  PROC DrawPart24()
    MoveL Offs(pOrigin,252.34,264.25,6.00),v60,z5,tPen\WObj:=wPaper;
    MoveL Offs(pOrigin,252.12,261.70,6.00),vTravel,z5,tPen\WObj:=wPaper;
    MoveL Offs(pOrigin,252.12,261.70,0.00),v60,z0,tPen\WObj:=wPaper;
    MoveL Offs(pOrigin,252.34,261.20,0.00),v40,z0,tPen\WObj:=wPaper;
    MoveL Offs(pOrigin,254.68,259.93,0.00),v40,z0,tPen\WObj:=wPaper;
    MoveL Offs(pOrigin,259.35,258.51,0.00),v40,z0,tPen\WObj:=wPaper;
    MoveL Offs(pOrigin,262.54,258.51,0.00),v40,fine,tPen\WObj:=wPaper;
    MoveL Offs(pOrigin,262.54,258.51,6.00),v60,z5,tPen\WObj:=wPaper;
    MoveL Offs(pOrigin,261.26,260.85,6.00),vTravel,z5,tPen\WObj:=wPaper;
    MoveL Offs(pOrigin,261.26,260.85,0.00),v60,z0,tPen\WObj:=wPaper;
    MoveL Offs(pOrigin,256.16,261.49,0.00),v40,z0,tPen\WObj:=wPaper;
    MoveL Offs(pOrigin,252.98,262.55,0.00),v40,z0,tPen\WObj:=wPaper;
    MoveL Offs(pOrigin,252.34,262.34,0.00),v40,z0,tPen\WObj:=wPaper;
    MoveL Offs(pOrigin,252.12,261.70,0.00),v40,fine,tPen\WObj:=wPaper;
    MoveL Offs(pOrigin,252.12,261.70,6.00),v60,z5,tPen\WObj:=wPaper;
    MoveL Offs(pOrigin,254.89,260.00,6.00),vTravel,z5,tPen\WObj:=wPaper;
    MoveL Offs(pOrigin,254.89,260.00,0.00),v60,z0,tPen\WObj:=wPaper;
    MoveL Offs(pOrigin,255.31,259.79,0.00),v40,z0,tPen\WObj:=wPaper;
    MoveL Offs(pOrigin,254.89,260.00,0.00),v40,fine,tPen\WObj:=wPaper;
    MoveL Offs(pOrigin,254.89,260.00,6.00),v60,z5,tPen\WObj:=wPaper;
    MoveL Offs(pOrigin,249.15,258.30,6.00),vTravel,z5,tPen\WObj:=wPaper;
    MoveL Offs(pOrigin,249.15,258.30,0.00),v60,z0,tPen\WObj:=wPaper;
    MoveL Offs(pOrigin,248.30,259.79,0.00),v40,z0,tPen\WObj:=wPaper;
    MoveL Offs(pOrigin,248.51,261.06,0.00),v40,fine,tPen\WObj:=wPaper;
    MoveL Offs(pOrigin,248.51,261.06,6.00),v60,z5,tPen\WObj:=wPaper;
    MoveL Offs(pOrigin,247.88,263.19,6.00),vTravel,z5,tPen\WObj:=wPaper;
    MoveL Offs(pOrigin,247.88,263.19,0.00),v60,z0,tPen\WObj:=wPaper;
    MoveL Offs(pOrigin,247.02,263.61,0.00),v40,z0,tPen\WObj:=wPaper;
    MoveL Offs(pOrigin,246.81,264.46,0.00),v40,z0,tPen\WObj:=wPaper;
    MoveL Offs(pOrigin,246.81,264.46,0.00),v40,z0,tPen\WObj:=wPaper;
    MoveL Offs(pOrigin,246.81,265.95,0.00),v40,z0,tPen\WObj:=wPaper;
    MoveL Offs(pOrigin,246.60,265.95,0.00),v40,z0,tPen\WObj:=wPaper;
    MoveL Offs(pOrigin,245.75,265.95,0.00),v40,z0,tPen\WObj:=wPaper;
    MoveL Offs(pOrigin,245.75,265.10,0.00),v40,z0,tPen\WObj:=wPaper;
    MoveL Offs(pOrigin,245.32,264.89,0.00),v40,z0,tPen\WObj:=wPaper;
    MoveL Offs(pOrigin,245.32,264.89,0.00),v40,z0,tPen\WObj:=wPaper;
    MoveL Offs(pOrigin,245.11,263.61,0.00),v40,z0,tPen\WObj:=wPaper;
    MoveL Offs(pOrigin,246.46,260.07,0.00),v40,z0,tPen\WObj:=wPaper;
    MoveL Offs(pOrigin,247.88,258.16,0.00),v40,z0,tPen\WObj:=wPaper;
    MoveL Offs(pOrigin,249.15,257.88,0.00),v40,fine,tPen\WObj:=wPaper;
    MoveL Offs(pOrigin,249.15,257.88,6.00),v60,z5,tPen\WObj:=wPaper;
    MoveL Offs(pOrigin,247.88,263.19,6.00),vTravel,z5,tPen\WObj:=wPaper;
    MoveL Offs(pOrigin,247.88,263.19,0.00),v60,z0,tPen\WObj:=wPaper;
    MoveL Offs(pOrigin,248.51,263.83,0.00),v40,fine,tPen\WObj:=wPaper;
    MoveL Offs(pOrigin,248.51,263.83,6.00),v60,z5,tPen\WObj:=wPaper;
    MoveL Offs(pOrigin,246.81,264.46,6.00),vTravel,z5,tPen\WObj:=wPaper;
    MoveL Offs(pOrigin,246.81,264.46,0.00),v60,z0,tPen\WObj:=wPaper;
    MoveL Offs(pOrigin,245.75,264.89,0.00),v40,z0,tPen\WObj:=wPaper;
    MoveL Offs(pOrigin,245.32,264.89,0.00),v40,z0,tPen\WObj:=wPaper;
    MoveL Offs(pOrigin,244.69,266.16,0.00),v40,z0,tPen\WObj:=wPaper;
    MoveL Offs(pOrigin,244.69,266.16,0.00),v40,z0,tPen\WObj:=wPaper;
    MoveL Offs(pOrigin,246.39,266.02,0.00),v40,z0,tPen\WObj:=wPaper;
    MoveL Offs(pOrigin,246.60,267.86,0.00),v40,z0,tPen\WObj:=wPaper;
    MoveL Offs(pOrigin,246.60,267.86,0.00),v40,z0,tPen\WObj:=wPaper;
    MoveL Offs(pOrigin,246.81,269.14,0.00),v40,z0,tPen\WObj:=wPaper;
    MoveL Offs(pOrigin,246.81,269.14,0.00),v40,z0,tPen\WObj:=wPaper;
    MoveL Offs(pOrigin,246.81,270.20,0.00),v40,z0,tPen\WObj:=wPaper;
    MoveL Offs(pOrigin,246.81,270.20,0.00),v40,z0,tPen\WObj:=wPaper;
    MoveL Offs(pOrigin,245.32,270.13,0.00),v40,z0,tPen\WObj:=wPaper;
    MoveL Offs(pOrigin,245.11,269.77,0.00),v40,z0,tPen\WObj:=wPaper;
    MoveL Offs(pOrigin,245.32,268.92,0.00),v40,z0,tPen\WObj:=wPaper;
    MoveL Offs(pOrigin,245.32,268.92,0.00),v40,z0,tPen\WObj:=wPaper;
    MoveL Offs(pOrigin,244.26,267.86,0.00),v40,z0,tPen\WObj:=wPaper;
    MoveL Offs(pOrigin,241.50,267.86,0.00),v40,z0,tPen\WObj:=wPaper;
    MoveL Offs(pOrigin,237.46,267.15,0.00),v40,z0,tPen\WObj:=wPaper;
    MoveL Offs(pOrigin,236.40,267.86,0.00),v40,z0,tPen\WObj:=wPaper;
    MoveL Offs(pOrigin,236.61,271.05,0.00),v40,z0,tPen\WObj:=wPaper;
    MoveL Offs(pOrigin,236.19,271.48,0.00),v40,fine,tPen\WObj:=wPaper;
    MoveL Offs(pOrigin,236.19,271.48,6.00),v60,z5,tPen\WObj:=wPaper;
    MoveL Offs(pOrigin,233.21,271.48,6.00),vTravel,z5,tPen\WObj:=wPaper;
    MoveL Offs(pOrigin,233.21,271.48,0.00),v60,z0,tPen\WObj:=wPaper;
    MoveL Offs(pOrigin,231.94,271.90,0.00),v40,z0,tPen\WObj:=wPaper;
    MoveL Offs(pOrigin,231.30,271.26,0.00),v40,z0,tPen\WObj:=wPaper;
    MoveL Offs(pOrigin,231.51,270.84,0.00),v40,z0,tPen\WObj:=wPaper;
    MoveL Offs(pOrigin,231.65,269.77,0.00),v40,z0,tPen\WObj:=wPaper;
    MoveL Offs(pOrigin,230.45,268.71,0.00),v40,z0,tPen\WObj:=wPaper;
    MoveL Offs(pOrigin,230.45,268.71,0.00),v40,z0,tPen\WObj:=wPaper;
    MoveL Offs(pOrigin,231.09,268.08,0.00),v40,z0,tPen\WObj:=wPaper;
    MoveL Offs(pOrigin,232.15,268.08,0.00),v40,z0,tPen\WObj:=wPaper;
    MoveL Offs(pOrigin,232.79,268.50,0.00),v40,z0,tPen\WObj:=wPaper;
    MoveL Offs(pOrigin,232.79,269.14,0.00),v40,z0,tPen\WObj:=wPaper;
    MoveL Offs(pOrigin,231.73,269.56,0.00),v40,fine,tPen\WObj:=wPaper;
    MoveL Offs(pOrigin,231.73,269.56,6.00),v60,z5,tPen\WObj:=wPaper;
    MoveL Offs(pOrigin,231.51,270.84,6.00),vTravel,z5,tPen\WObj:=wPaper;
    MoveL Offs(pOrigin,231.51,270.84,0.00),v60,z0,tPen\WObj:=wPaper;
    MoveL Offs(pOrigin,233.21,270.84,0.00),v40,z0,tPen\WObj:=wPaper;
    MoveL Offs(pOrigin,233.21,270.84,0.00),v40,z0,tPen\WObj:=wPaper;
    MoveL Offs(pOrigin,233.00,268.57,0.00),v40,z0,tPen\WObj:=wPaper;
    MoveL Offs(pOrigin,234.06,268.22,0.00),v40,z0,tPen\WObj:=wPaper;
    MoveL Offs(pOrigin,235.48,269.14,0.00),v40,z0,tPen\WObj:=wPaper;
    MoveL Offs(pOrigin,236.19,271.90,0.00),v40,z0,tPen\WObj:=wPaper;
    MoveL Offs(pOrigin,236.19,275.30,0.00),v40,fine,tPen\WObj:=wPaper;
    MoveL Offs(pOrigin,236.19,275.30,6.00),v60,z5,tPen\WObj:=wPaper;
    MoveL Offs(pOrigin,231.73,271.90,6.00),vTravel,z5,tPen\WObj:=wPaper;
    MoveL Offs(pOrigin,231.73,271.90,0.00),v60,z0,tPen\WObj:=wPaper;
    MoveL Offs(pOrigin,230.88,271.26,0.00),v40,z0,tPen\WObj:=wPaper;
    MoveL Offs(pOrigin,226.41,271.69,0.00),v40,z0,tPen\WObj:=wPaper;
    MoveL Offs(pOrigin,217.49,270.41,0.00),v40,z0,tPen\WObj:=wPaper;
    MoveL Offs(pOrigin,217.13,270.62,0.00),v40,z0,tPen\WObj:=wPaper;
    MoveL Offs(pOrigin,217.27,271.05,0.00),v40,z0,tPen\WObj:=wPaper;
    MoveL Offs(pOrigin,217.06,270.41,0.00),v40,z0,tPen\WObj:=wPaper;
    MoveL Offs(pOrigin,214.30,268.57,0.00),v40,z0,tPen\WObj:=wPaper;
    MoveL Offs(pOrigin,213.88,267.86,0.00),v40,z0,tPen\WObj:=wPaper;
    MoveL Offs(pOrigin,213.88,267.86,0.00),v40,z0,tPen\WObj:=wPaper;
    MoveL Offs(pOrigin,214.73,267.65,0.00),v40,z0,tPen\WObj:=wPaper;
    MoveL Offs(pOrigin,215.15,268.71,0.00),v40,z0,tPen\WObj:=wPaper;
    MoveL Offs(pOrigin,215.15,268.08,0.00),v40,z0,tPen\WObj:=wPaper;
    MoveL Offs(pOrigin,219.19,268.50,0.00),v40,z0,tPen\WObj:=wPaper;
    MoveL Offs(pOrigin,219.19,268.50,0.00),v40,z0,tPen\WObj:=wPaper;
    MoveL Offs(pOrigin,222.38,268.92,0.00),v40,z0,tPen\WObj:=wPaper;
    MoveL Offs(pOrigin,222.38,268.92,0.00),v40,z0,tPen\WObj:=wPaper;
    MoveL Offs(pOrigin,225.56,269.14,0.00),v40,z0,tPen\WObj:=wPaper;
    MoveL Offs(pOrigin,225.56,269.14,0.00),v40,z0,tPen\WObj:=wPaper;
    MoveL Offs(pOrigin,228.96,269.35,0.00),v40,z0,tPen\WObj:=wPaper;
    MoveL Offs(pOrigin,229.81,268.71,0.00),v40,z0,tPen\WObj:=wPaper;
    MoveL Offs(pOrigin,230.45,268.71,0.00),v40,z0,tPen\WObj:=wPaper;
    MoveL Offs(pOrigin,229.60,268.50,0.00),v40,z0,tPen\WObj:=wPaper;
    MoveL Offs(pOrigin,229.18,267.65,0.00),v40,z0,tPen\WObj:=wPaper;
    MoveL Offs(pOrigin,229.18,267.65,0.00),v40,z0,tPen\WObj:=wPaper;
    MoveL Offs(pOrigin,225.14,267.44,0.00),v40,z0,tPen\WObj:=wPaper;
  ENDPROC

  PROC DrawPart25()
    MoveL Offs(pOrigin,223.23,267.01,0.00),v40,z0,tPen\WObj:=wPaper;
    MoveL Offs(pOrigin,222.52,268.08,0.00),v40,z0,tPen\WObj:=wPaper;
    MoveL Offs(pOrigin,225.56,268.50,0.00),v40,z0,tPen\WObj:=wPaper;
    MoveL Offs(pOrigin,225.56,268.50,0.00),v40,z0,tPen\WObj:=wPaper;
    MoveL Offs(pOrigin,229.18,268.29,0.00),v40,z0,tPen\WObj:=wPaper;
    MoveL Offs(pOrigin,229.18,267.65,0.00),v40,z0,tPen\WObj:=wPaper;
    MoveL Offs(pOrigin,229.81,267.01,0.00),v40,z0,tPen\WObj:=wPaper;
    MoveL Offs(pOrigin,229.81,267.01,0.00),v40,z0,tPen\WObj:=wPaper;
    MoveL Offs(pOrigin,229.18,266.59,0.00),v40,z0,tPen\WObj:=wPaper;
    MoveL Offs(pOrigin,228.11,266.59,0.00),v40,z0,tPen\WObj:=wPaper;
    MoveL Offs(pOrigin,222.38,264.75,0.00),v40,z0,tPen\WObj:=wPaper;
    MoveL Offs(pOrigin,220.46,263.90,0.00),v40,z0,tPen\WObj:=wPaper;
    MoveL Offs(pOrigin,218.76,262.76,0.00),v40,z0,tPen\WObj:=wPaper;
    MoveL Offs(pOrigin,218.34,262.12,0.00),v40,z0,tPen\WObj:=wPaper;
    MoveL Offs(pOrigin,218.34,262.12,0.00),v40,z0,tPen\WObj:=wPaper;
    MoveL Offs(pOrigin,217.06,261.49,0.00),v40,z0,tPen\WObj:=wPaper;
    MoveL Offs(pOrigin,216.21,259.58,0.00),v40,z0,tPen\WObj:=wPaper;
    MoveL Offs(pOrigin,216.21,259.58,0.00),v40,z0,tPen\WObj:=wPaper;
    MoveL Offs(pOrigin,217.27,259.15,0.00),v40,z0,tPen\WObj:=wPaper;
    MoveL Offs(pOrigin,218.55,259.93,0.00),v40,z0,tPen\WObj:=wPaper;
    MoveL Offs(pOrigin,219.82,260.00,0.00),v40,z0,tPen\WObj:=wPaper;
    MoveL Offs(pOrigin,219.82,260.00,0.00),v40,z0,tPen\WObj:=wPaper;
    MoveL Offs(pOrigin,219.82,260.64,0.00),v40,z0,tPen\WObj:=wPaper;
    MoveL Offs(pOrigin,220.68,260.64,0.00),v40,z0,tPen\WObj:=wPaper;
    MoveL Offs(pOrigin,220.68,260.64,0.00),v40,z0,tPen\WObj:=wPaper;
    MoveL Offs(pOrigin,220.46,259.79,0.00),v40,z0,tPen\WObj:=wPaper;
    MoveL Offs(pOrigin,219.82,260.00,0.00),v40,z0,tPen\WObj:=wPaper;
    MoveL Offs(pOrigin,220.68,259.79,0.00),v40,z0,tPen\WObj:=wPaper;
    MoveL Offs(pOrigin,222.80,259.36,0.00),v40,z0,tPen\WObj:=wPaper;
    MoveL Offs(pOrigin,223.01,260.42,0.00),v40,z0,tPen\WObj:=wPaper;
    MoveL Offs(pOrigin,221.10,260.71,0.00),v40,z0,tPen\WObj:=wPaper;
    MoveL Offs(pOrigin,220.89,261.49,0.00),v40,z0,tPen\WObj:=wPaper;
    MoveL Offs(pOrigin,221.10,261.91,0.00),v40,z0,tPen\WObj:=wPaper;
    MoveL Offs(pOrigin,222.80,262.83,0.00),v40,z0,tPen\WObj:=wPaper;
    MoveL Offs(pOrigin,223.08,262.20,0.00),v40,z0,tPen\WObj:=wPaper;
    MoveL Offs(pOrigin,224.07,261.49,0.00),v40,z0,tPen\WObj:=wPaper;
    MoveL Offs(pOrigin,224.07,260.85,0.00),v40,z0,tPen\WObj:=wPaper;
    MoveL Offs(pOrigin,225.99,260.64,0.00),v40,z0,tPen\WObj:=wPaper;
    MoveL Offs(pOrigin,226.20,261.06,0.00),v40,z0,tPen\WObj:=wPaper;
    MoveL Offs(pOrigin,226.20,261.06,0.00),v40,z0,tPen\WObj:=wPaper;
    MoveL Offs(pOrigin,227.05,261.27,0.00),v40,z0,tPen\WObj:=wPaper;
    MoveL Offs(pOrigin,227.69,262.12,0.00),v40,z0,tPen\WObj:=wPaper;
    MoveL Offs(pOrigin,227.69,263.40,0.00),v40,fine,tPen\WObj:=wPaper;
    MoveL Offs(pOrigin,227.69,263.40,6.00),v60,z5,tPen\WObj:=wPaper;
    MoveL Offs(pOrigin,227.90,262.12,6.00),vTravel,z5,tPen\WObj:=wPaper;
    MoveL Offs(pOrigin,227.90,262.12,0.00),v60,z0,tPen\WObj:=wPaper;
    MoveL Offs(pOrigin,228.96,261.91,0.00),v40,z0,tPen\WObj:=wPaper;
    MoveL Offs(pOrigin,228.96,261.91,0.00),v40,z0,tPen\WObj:=wPaper;
    MoveL Offs(pOrigin,229.60,263.61,0.00),v40,z0,tPen\WObj:=wPaper;
    MoveL Offs(pOrigin,230.88,263.26,0.00),v40,z0,tPen\WObj:=wPaper;
    MoveL Offs(pOrigin,231.51,262.34,0.00),v40,z0,tPen\WObj:=wPaper;
    MoveL Offs(pOrigin,231.51,262.34,0.00),v40,z0,tPen\WObj:=wPaper;
    MoveL Offs(pOrigin,233.21,262.12,0.00),v40,z0,tPen\WObj:=wPaper;
    MoveL Offs(pOrigin,233.21,262.12,0.00),v40,z0,tPen\WObj:=wPaper;
    MoveL Offs(pOrigin,233.64,262.98,0.00),v40,fine,tPen\WObj:=wPaper;
    MoveL Offs(pOrigin,233.64,262.98,6.00),v60,z5,tPen\WObj:=wPaper;
    MoveL Offs(pOrigin,233.85,264.46,6.00),vTravel,z5,tPen\WObj:=wPaper;
    MoveL Offs(pOrigin,233.85,264.46,0.00),v60,z0,tPen\WObj:=wPaper;
    MoveL Offs(pOrigin,234.84,263.54,0.00),v40,z0,tPen\WObj:=wPaper;
    MoveL Offs(pOrigin,234.91,262.83,0.00),v40,z0,tPen\WObj:=wPaper;
    MoveL Offs(pOrigin,233.85,262.98,0.00),v40,z0,tPen\WObj:=wPaper;
    MoveL Offs(pOrigin,233.28,263.61,0.00),v40,z0,tPen\WObj:=wPaper;
    MoveL Offs(pOrigin,233.21,264.46,0.00),v40,z0,tPen\WObj:=wPaper;
    MoveL Offs(pOrigin,233.21,264.46,0.00),v40,z0,tPen\WObj:=wPaper;
    MoveL Offs(pOrigin,234.27,264.89,0.00),v40,z0,tPen\WObj:=wPaper;
    MoveL Offs(pOrigin,235.34,265.95,0.00),v40,z0,tPen\WObj:=wPaper;
    MoveL Offs(pOrigin,235.27,267.23,0.00),v40,z0,tPen\WObj:=wPaper;
    MoveL Offs(pOrigin,234.27,268.08,0.00),v40,z0,tPen\WObj:=wPaper;
    MoveL Offs(pOrigin,233.85,268.08,0.00),v40,z0,tPen\WObj:=wPaper;
    MoveL Offs(pOrigin,233.14,266.87,0.00),v40,z0,tPen\WObj:=wPaper;
    MoveL Offs(pOrigin,231.51,266.59,0.00),v40,z0,tPen\WObj:=wPaper;
    MoveL Offs(pOrigin,231.51,266.59,0.00),v40,z0,tPen\WObj:=wPaper;
    MoveL Offs(pOrigin,230.45,267.01,0.00),v40,z0,tPen\WObj:=wPaper;
    MoveL Offs(pOrigin,230.45,267.01,0.00),v40,z0,tPen\WObj:=wPaper;
    MoveL Offs(pOrigin,230.66,268.08,0.00),v40,fine,tPen\WObj:=wPaper;
    MoveL Offs(pOrigin,230.66,268.08,6.00),v60,z5,tPen\WObj:=wPaper;
    MoveL Offs(pOrigin,231.51,266.59,6.00),vTravel,z5,tPen\WObj:=wPaper;
    MoveL Offs(pOrigin,231.51,266.59,0.00),v60,z0,tPen\WObj:=wPaper;
    MoveL Offs(pOrigin,232.36,265.74,0.00),v40,z0,tPen\WObj:=wPaper;
    MoveL Offs(pOrigin,232.79,264.46,0.00),v40,z0,tPen\WObj:=wPaper;
    MoveL Offs(pOrigin,232.79,264.46,0.00),v40,z0,tPen\WObj:=wPaper;
    MoveL Offs(pOrigin,232.15,264.25,0.00),v40,z0,tPen\WObj:=wPaper;
    MoveL Offs(pOrigin,230.45,264.89,0.00),v40,z0,tPen\WObj:=wPaper;
    MoveL Offs(pOrigin,230.38,264.89,0.00),v40,z0,tPen\WObj:=wPaper;
    MoveL Offs(pOrigin,230.17,265.45,0.00),v40,z0,tPen\WObj:=wPaper;
    MoveL Offs(pOrigin,229.39,265.74,0.00),v40,z0,tPen\WObj:=wPaper;
    MoveL Offs(pOrigin,228.40,265.52,0.00),v40,z0,tPen\WObj:=wPaper;
    MoveL Offs(pOrigin,228.96,264.89,0.00),v40,z0,tPen\WObj:=wPaper;
    MoveL Offs(pOrigin,229.81,264.67,0.00),v40,z0,tPen\WObj:=wPaper;
    MoveL Offs(pOrigin,230.38,264.89,0.00),v40,fine,tPen\WObj:=wPaper;
    MoveL Offs(pOrigin,230.38,264.89,6.00),v60,z5,tPen\WObj:=wPaper;
    MoveL Offs(pOrigin,228.32,265.10,6.00),vTravel,z5,tPen\WObj:=wPaper;
    MoveL Offs(pOrigin,228.32,265.10,0.00),v60,z0,tPen\WObj:=wPaper;
    MoveL Offs(pOrigin,226.84,265.10,0.00),v40,z0,tPen\WObj:=wPaper;
    MoveL Offs(pOrigin,226.41,265.74,0.00),v40,fine,tPen\WObj:=wPaper;
    MoveL Offs(pOrigin,226.41,265.74,6.00),v60,z5,tPen\WObj:=wPaper;
    MoveL Offs(pOrigin,222.80,267.01,6.00),vTravel,z5,tPen\WObj:=wPaper;
    MoveL Offs(pOrigin,222.80,267.01,0.00),v60,z0,tPen\WObj:=wPaper;
    MoveL Offs(pOrigin,221.74,266.80,0.00),v40,z0,tPen\WObj:=wPaper;
    MoveL Offs(pOrigin,221.52,267.23,0.00),v40,z0,tPen\WObj:=wPaper;
    MoveL Offs(pOrigin,221.52,267.23,0.00),v40,z0,tPen\WObj:=wPaper;
    MoveL Offs(pOrigin,217.49,266.09,0.00),v40,z0,tPen\WObj:=wPaper;
    MoveL Offs(pOrigin,215.15,264.67,0.00),v40,z0,tPen\WObj:=wPaper;
    MoveL Offs(pOrigin,214.73,263.90,0.00),v40,z0,tPen\WObj:=wPaper;
    MoveL Offs(pOrigin,213.88,263.68,0.00),v40,z0,tPen\WObj:=wPaper;
    MoveL Offs(pOrigin,213.24,262.98,0.00),v40,z0,tPen\WObj:=wPaper;
    MoveL Offs(pOrigin,213.24,262.98,0.00),v40,z0,tPen\WObj:=wPaper;
    MoveL Offs(pOrigin,212.67,260.42,0.00),v40,z0,tPen\WObj:=wPaper;
    MoveL Offs(pOrigin,214.51,259.15,0.00),v40,z0,tPen\WObj:=wPaper;
    MoveL Offs(pOrigin,214.51,259.15,0.00),v40,z0,tPen\WObj:=wPaper;
    MoveL Offs(pOrigin,213.66,258.51,0.00),v40,z0,tPen\WObj:=wPaper;
    MoveL Offs(pOrigin,211.75,258.51,0.00),v40,fine,tPen\WObj:=wPaper;
    MoveL Offs(pOrigin,211.75,258.51,6.00),v60,z5,tPen\WObj:=wPaper;
    MoveL Offs(pOrigin,213.45,256.60,6.00),vTravel,z5,tPen\WObj:=wPaper;
    MoveL Offs(pOrigin,213.45,256.60,0.00),v60,z0,tPen\WObj:=wPaper;
    MoveL Offs(pOrigin,214.73,257.45,0.00),v40,z0,tPen\WObj:=wPaper;
    MoveL Offs(pOrigin,215.36,259.15,0.00),v40,z0,tPen\WObj:=wPaper;
    MoveL Offs(pOrigin,215.36,259.15,0.00),v40,z0,tPen\WObj:=wPaper;
    MoveL Offs(pOrigin,216.21,259.58,0.00),v40,fine,tPen\WObj:=wPaper;
    MoveL Offs(pOrigin,216.21,259.58,6.00),v60,z5,tPen\WObj:=wPaper;
  ENDPROC

  PROC DrawPart26()
    MoveL Offs(pOrigin,217.91,259.58,6.00),vTravel,z5,tPen\WObj:=wPaper;
    MoveL Offs(pOrigin,217.91,259.58,0.00),v60,z0,tPen\WObj:=wPaper;
    MoveL Offs(pOrigin,218.34,260.00,0.00),v40,z0,tPen\WObj:=wPaper;
    MoveL Offs(pOrigin,217.91,259.58,0.00),v40,fine,tPen\WObj:=wPaper;
    MoveL Offs(pOrigin,217.91,259.58,6.00),v60,z5,tPen\WObj:=wPaper;
    MoveL Offs(pOrigin,216.85,261.49,6.00),vTravel,z5,tPen\WObj:=wPaper;
    MoveL Offs(pOrigin,216.85,261.49,0.00),v60,z0,tPen\WObj:=wPaper;
    MoveL Offs(pOrigin,217.27,261.91,0.00),v40,z0,tPen\WObj:=wPaper;
    MoveL Offs(pOrigin,216.85,261.49,0.00),v40,fine,tPen\WObj:=wPaper;
    MoveL Offs(pOrigin,216.85,261.49,6.00),v60,z5,tPen\WObj:=wPaper;
    MoveL Offs(pOrigin,215.79,265.31,6.00),vTravel,z5,tPen\WObj:=wPaper;
    MoveL Offs(pOrigin,215.79,265.31,0.00),v60,z0,tPen\WObj:=wPaper;
    MoveL Offs(pOrigin,216.21,265.52,0.00),v40,z0,tPen\WObj:=wPaper;
    MoveL Offs(pOrigin,215.79,265.31,0.00),v40,fine,tPen\WObj:=wPaper;
    MoveL Offs(pOrigin,215.79,265.31,6.00),v60,z5,tPen\WObj:=wPaper;
    MoveL Offs(pOrigin,213.88,267.86,6.00),vTravel,z5,tPen\WObj:=wPaper;
    MoveL Offs(pOrigin,213.88,267.86,0.00),v60,z0,tPen\WObj:=wPaper;
    MoveL Offs(pOrigin,209.41,266.30,0.00),v40,z0,tPen\WObj:=wPaper;
    MoveL Offs(pOrigin,208.77,265.17,0.00),v40,z0,tPen\WObj:=wPaper;
    MoveL Offs(pOrigin,207.57,264.67,0.00),v40,z0,tPen\WObj:=wPaper;
    MoveL Offs(pOrigin,207.29,263.61,0.00),v40,z0,tPen\WObj:=wPaper;
    MoveL Offs(pOrigin,207.29,263.61,0.00),v40,z0,tPen\WObj:=wPaper;
    MoveL Offs(pOrigin,204.52,263.12,0.00),v40,z0,tPen\WObj:=wPaper;
    MoveL Offs(pOrigin,204.10,261.91,0.00),v40,z0,tPen\WObj:=wPaper;
    MoveL Offs(pOrigin,204.10,261.91,0.00),v40,z0,tPen\WObj:=wPaper;
    MoveL Offs(pOrigin,207.07,260.92,0.00),v40,z0,tPen\WObj:=wPaper;
    MoveL Offs(pOrigin,207.29,263.61,0.00),v40,fine,tPen\WObj:=wPaper;
    MoveL Offs(pOrigin,207.29,263.61,6.00),v60,z5,tPen\WObj:=wPaper;
    MoveL Offs(pOrigin,207.50,265.31,6.00),vTravel,z5,tPen\WObj:=wPaper;
    MoveL Offs(pOrigin,207.50,265.31,0.00),v60,z0,tPen\WObj:=wPaper;
    MoveL Offs(pOrigin,206.65,265.95,0.00),v40,z0,tPen\WObj:=wPaper;
    MoveL Offs(pOrigin,206.23,270.84,0.00),v40,z0,tPen\WObj:=wPaper;
    MoveL Offs(pOrigin,205.38,272.33,0.00),v40,z0,tPen\WObj:=wPaper;
    MoveL Offs(pOrigin,205.30,274.45,0.00),v40,z0,tPen\WObj:=wPaper;
    MoveL Offs(pOrigin,204.74,275.09,0.00),v40,z0,tPen\WObj:=wPaper;
    MoveL Offs(pOrigin,204.88,276.72,0.00),v40,z0,tPen\WObj:=wPaper;
    MoveL Offs(pOrigin,204.31,277.21,0.00),v40,z0,tPen\WObj:=wPaper;
    MoveL Offs(pOrigin,204.52,279.12,0.00),v40,z0,tPen\WObj:=wPaper;
    MoveL Offs(pOrigin,204.52,279.12,0.00),v40,z0,tPen\WObj:=wPaper;
    MoveL Offs(pOrigin,203.75,279.76,0.00),v40,z0,tPen\WObj:=wPaper;
    MoveL Offs(pOrigin,203.53,280.83,0.00),v40,z0,tPen\WObj:=wPaper;
    MoveL Offs(pOrigin,204.17,281.46,0.00),v40,z0,tPen\WObj:=wPaper;
    MoveL Offs(pOrigin,204.74,282.95,0.00),v40,z0,tPen\WObj:=wPaper;
    MoveL Offs(pOrigin,204.95,284.86,0.00),v40,z0,tPen\WObj:=wPaper;
    MoveL Offs(pOrigin,204.74,286.56,0.00),v40,z0,tPen\WObj:=wPaper;
    MoveL Offs(pOrigin,204.74,286.56,0.00),v40,z0,tPen\WObj:=wPaper;
    MoveL Offs(pOrigin,205.45,289.11,0.00),v40,z0,tPen\WObj:=wPaper;
    MoveL Offs(pOrigin,206.65,290.17,0.00),v40,z0,tPen\WObj:=wPaper;
    MoveL Offs(pOrigin,206.23,291.24,0.00),v40,z0,tPen\WObj:=wPaper;
    MoveL Offs(pOrigin,206.23,291.24,0.00),v40,z0,tPen\WObj:=wPaper;
    MoveL Offs(pOrigin,206.23,293.15,0.00),v40,fine,tPen\WObj:=wPaper;
    MoveL Offs(pOrigin,206.23,293.15,6.00),v60,z5,tPen\WObj:=wPaper;
    MoveL Offs(pOrigin,206.23,291.24,6.00),vTravel,z5,tPen\WObj:=wPaper;
    MoveL Offs(pOrigin,206.23,291.24,0.00),v60,z0,tPen\WObj:=wPaper;
    MoveL Offs(pOrigin,205.38,290.81,0.00),v40,z0,tPen\WObj:=wPaper;
    MoveL Offs(pOrigin,205.16,290.17,0.00),v40,z0,tPen\WObj:=wPaper;
    MoveL Offs(pOrigin,205.38,289.33,0.00),v40,z0,tPen\WObj:=wPaper;
    MoveL Offs(pOrigin,205.80,289.54,0.00),v40,z0,tPen\WObj:=wPaper;
    MoveL Offs(pOrigin,206.23,289.75,0.00),v40,z0,tPen\WObj:=wPaper;
    MoveL Offs(pOrigin,205.80,289.54,0.00),v40,fine,tPen\WObj:=wPaper;
    MoveL Offs(pOrigin,205.80,289.54,6.00),v60,z5,tPen\WObj:=wPaper;
    MoveL Offs(pOrigin,202.40,289.96,6.00),vTravel,z5,tPen\WObj:=wPaper;
    MoveL Offs(pOrigin,202.40,289.96,0.00),v60,z0,tPen\WObj:=wPaper;
    MoveL Offs(pOrigin,202.40,289.11,0.00),v40,z0,tPen\WObj:=wPaper;
    MoveL Offs(pOrigin,201.55,288.69,0.00),v40,z0,tPen\WObj:=wPaper;
    MoveL Offs(pOrigin,201.55,288.69,0.00),v40,z0,tPen\WObj:=wPaper;
    MoveL Offs(pOrigin,200.35,286.14,0.00),v40,z0,tPen\WObj:=wPaper;
    MoveL Offs(pOrigin,199.21,284.79,0.00),v40,z0,tPen\WObj:=wPaper;
    MoveL Offs(pOrigin,198.36,284.44,0.00),v40,z0,tPen\WObj:=wPaper;
    MoveL Offs(pOrigin,197.37,285.29,0.00),v40,z0,tPen\WObj:=wPaper;
    MoveL Offs(pOrigin,197.30,286.14,0.00),v40,z0,tPen\WObj:=wPaper;
    MoveL Offs(pOrigin,197.30,286.14,0.00),v40,z0,tPen\WObj:=wPaper;
    MoveL Offs(pOrigin,197.44,287.20,0.00),v40,z0,tPen\WObj:=wPaper;
    MoveL Offs(pOrigin,199.07,289.96,0.00),v40,z0,tPen\WObj:=wPaper;
    MoveL Offs(pOrigin,199.43,291.45,0.00),v40,z0,tPen\WObj:=wPaper;
    MoveL Offs(pOrigin,199.43,291.45,0.00),v40,z0,tPen\WObj:=wPaper;
    MoveL Offs(pOrigin,198.01,290.81,0.00),v40,z0,tPen\WObj:=wPaper;
    MoveL Offs(pOrigin,195.74,286.35,0.00),v40,z0,tPen\WObj:=wPaper;
    MoveL Offs(pOrigin,195.18,285.92,0.00),v40,z0,tPen\WObj:=wPaper;
    MoveL Offs(pOrigin,195.18,285.92,0.00),v40,z0,tPen\WObj:=wPaper;
    MoveL Offs(pOrigin,194.54,287.20,0.00),v40,z0,tPen\WObj:=wPaper;
    MoveL Offs(pOrigin,193.90,287.20,0.00),v40,z0,tPen\WObj:=wPaper;
    MoveL Offs(pOrigin,193.26,287.84,0.00),v40,z0,tPen\WObj:=wPaper;
    MoveL Offs(pOrigin,193.69,289.11,0.00),v40,z0,tPen\WObj:=wPaper;
    MoveL Offs(pOrigin,194.32,289.89,0.00),v40,z0,tPen\WObj:=wPaper;
    MoveL Offs(pOrigin,195.10,290.25,0.00),v40,z0,tPen\WObj:=wPaper;
    MoveL Offs(pOrigin,199.21,295.91,0.00),v40,z0,tPen\WObj:=wPaper;
    MoveL Offs(pOrigin,200.91,297.47,0.00),v40,z0,tPen\WObj:=wPaper;
    MoveL Offs(pOrigin,201.98,297.61,0.00),v40,z0,tPen\WObj:=wPaper;
    MoveL Offs(pOrigin,201.98,297.61,0.00),v40,z0,tPen\WObj:=wPaper;
    MoveL Offs(pOrigin,201.98,296.55,0.00),v40,z0,tPen\WObj:=wPaper;
    MoveL Offs(pOrigin,201.98,296.55,0.00),v40,z0,tPen\WObj:=wPaper;
    MoveL Offs(pOrigin,204.10,296.12,0.00),v40,z0,tPen\WObj:=wPaper;
    MoveL Offs(pOrigin,204.10,296.12,0.00),v40,z0,tPen\WObj:=wPaper;
    MoveL Offs(pOrigin,203.82,295.06,0.00),v40,z0,tPen\WObj:=wPaper;
    MoveL Offs(pOrigin,203.25,294.42,0.00),v40,z0,tPen\WObj:=wPaper;
    MoveL Offs(pOrigin,201.55,293.79,0.00),v40,z0,tPen\WObj:=wPaper;
    MoveL Offs(pOrigin,201.12,294.21,0.00),v40,z0,tPen\WObj:=wPaper;
    MoveL Offs(pOrigin,201.98,296.55,0.00),v40,z0,tPen\WObj:=wPaper;
    MoveL Offs(pOrigin,201.98,297.61,0.00),v40,z0,tPen\WObj:=wPaper;
    MoveL Offs(pOrigin,202.40,298.46,0.00),v40,fine,tPen\WObj:=wPaper;
    MoveL Offs(pOrigin,202.40,298.46,6.00),v60,z5,tPen\WObj:=wPaper;
    MoveL Offs(pOrigin,202.40,299.95,6.00),vTravel,z5,tPen\WObj:=wPaper;
    MoveL Offs(pOrigin,202.40,299.95,0.00),v60,z0,tPen\WObj:=wPaper;
    MoveL Offs(pOrigin,200.49,299.31,0.00),v40,z0,tPen\WObj:=wPaper;
    MoveL Offs(pOrigin,199.71,299.52,0.00),v40,z0,tPen\WObj:=wPaper;
    MoveL Offs(pOrigin,199.71,300.38,0.00),v40,z0,tPen\WObj:=wPaper;
    MoveL Offs(pOrigin,201.34,301.86,0.00),v40,z0,tPen\WObj:=wPaper;
    MoveL Offs(pOrigin,201.34,301.86,0.00),v40,z0,tPen\WObj:=wPaper;
    MoveL Offs(pOrigin,201.34,302.92,0.00),v40,z0,tPen\WObj:=wPaper;
    MoveL Offs(pOrigin,201.34,302.92,0.00),v40,z0,tPen\WObj:=wPaper;
    MoveL Offs(pOrigin,203.04,303.92,0.00),v40,z0,tPen\WObj:=wPaper;
    MoveL Offs(pOrigin,204.74,304.41,0.00),v40,fine,tPen\WObj:=wPaper;
    MoveL Offs(pOrigin,204.74,304.41,6.00),v60,z5,tPen\WObj:=wPaper;
    MoveL Offs(pOrigin,204.74,306.11,6.00),vTravel,z5,tPen\WObj:=wPaper;
    MoveL Offs(pOrigin,204.74,306.11,0.00),v60,z0,tPen\WObj:=wPaper;
    MoveL Offs(pOrigin,204.31,305.55,0.00),v40,z0,tPen\WObj:=wPaper;
    MoveL Offs(pOrigin,200.27,304.27,0.00),v40,z0,tPen\WObj:=wPaper;
    MoveL Offs(pOrigin,198.36,302.71,0.00),v40,z0,tPen\WObj:=wPaper;
    MoveL Offs(pOrigin,196.66,301.86,0.00),v40,z0,tPen\WObj:=wPaper;
  ENDPROC

  PROC DrawPart27()
    MoveL Offs(pOrigin,194.47,298.46,0.00),v40,z0,tPen\WObj:=wPaper;
    MoveL Offs(pOrigin,193.90,298.04,0.00),v40,z0,tPen\WObj:=wPaper;
    MoveL Offs(pOrigin,193.90,298.04,0.00),v40,z0,tPen\WObj:=wPaper;
    MoveL Offs(pOrigin,193.69,298.67,0.00),v40,z0,tPen\WObj:=wPaper;
    MoveL Offs(pOrigin,194.68,301.44,0.00),v40,z0,tPen\WObj:=wPaper;
    MoveL Offs(pOrigin,196.88,304.84,0.00),v40,z0,tPen\WObj:=wPaper;
    MoveL Offs(pOrigin,200.06,306.47,0.00),v40,z0,tPen\WObj:=wPaper;
    MoveL Offs(pOrigin,200.91,306.25,0.00),v40,z0,tPen\WObj:=wPaper;
    MoveL Offs(pOrigin,203.25,306.75,0.00),v40,z0,tPen\WObj:=wPaper;
    MoveL Offs(pOrigin,203.25,306.75,0.00),v40,z0,tPen\WObj:=wPaper;
    MoveL Offs(pOrigin,204.10,307.81,0.00),v40,z0,tPen\WObj:=wPaper;
    MoveL Offs(pOrigin,203.89,308.45,0.00),v40,z0,tPen\WObj:=wPaper;
    MoveL Offs(pOrigin,204.52,307.81,0.00),v40,z0,tPen\WObj:=wPaper;
    MoveL Offs(pOrigin,206.86,307.60,0.00),v40,fine,tPen\WObj:=wPaper;
    MoveL Offs(pOrigin,206.86,307.60,6.00),v60,z5,tPen\WObj:=wPaper;
    MoveL Offs(pOrigin,208.35,306.11,6.00),vTravel,z5,tPen\WObj:=wPaper;
    MoveL Offs(pOrigin,208.35,306.11,0.00),v60,z0,tPen\WObj:=wPaper;
    MoveL Offs(pOrigin,204.74,306.11,0.00),v40,z0,tPen\WObj:=wPaper;
    MoveL Offs(pOrigin,204.74,306.11,0.00),v40,z0,tPen\WObj:=wPaper;
    MoveL Offs(pOrigin,203.68,306.33,0.00),v40,z0,tPen\WObj:=wPaper;
    MoveL Offs(pOrigin,203.25,306.75,0.00),v40,fine,tPen\WObj:=wPaper;
    MoveL Offs(pOrigin,203.25,306.75,6.00),v60,z5,tPen\WObj:=wPaper;
    MoveL Offs(pOrigin,204.74,309.09,6.00),vTravel,z5,tPen\WObj:=wPaper;
    MoveL Offs(pOrigin,204.74,309.09,0.00),v60,z0,tPen\WObj:=wPaper;
    MoveL Offs(pOrigin,205.38,309.94,0.00),v40,z0,tPen\WObj:=wPaper;
    MoveL Offs(pOrigin,205.38,309.94,0.00),v40,z0,tPen\WObj:=wPaper;
    MoveL Offs(pOrigin,203.68,308.52,0.00),v40,z0,tPen\WObj:=wPaper;
    MoveL Offs(pOrigin,200.27,308.24,0.00),v40,z0,tPen\WObj:=wPaper;
    MoveL Offs(pOrigin,197.73,307.32,0.00),v40,z0,tPen\WObj:=wPaper;
    MoveL Offs(pOrigin,195.18,305.69,0.00),v40,z0,tPen\WObj:=wPaper;
    MoveL Offs(pOrigin,194.32,304.20,0.00),v40,z0,tPen\WObj:=wPaper;
    MoveL Offs(pOrigin,193.90,303.99,0.00),v40,z0,tPen\WObj:=wPaper;
    MoveL Offs(pOrigin,193.90,303.99,0.00),v40,z0,tPen\WObj:=wPaper;
    MoveL Offs(pOrigin,193.26,300.16,0.00),v40,fine,tPen\WObj:=wPaper;
    MoveL Offs(pOrigin,193.26,300.16,6.00),v60,z5,tPen\WObj:=wPaper;
    MoveL Offs(pOrigin,191.35,300.80,6.00),vTravel,z5,tPen\WObj:=wPaper;
    MoveL Offs(pOrigin,191.35,300.80,0.00),v60,z0,tPen\WObj:=wPaper;
    MoveL Offs(pOrigin,191.35,296.98,0.00),v40,z0,tPen\WObj:=wPaper;
    MoveL Offs(pOrigin,192.41,293.58,0.00),v40,z0,tPen\WObj:=wPaper;
    MoveL Offs(pOrigin,191.63,292.73,0.00),v40,z0,tPen\WObj:=wPaper;
    MoveL Offs(pOrigin,191.49,291.95,0.00),v40,z0,tPen\WObj:=wPaper;
    MoveL Offs(pOrigin,190.93,291.66,0.00),v40,z0,tPen\WObj:=wPaper;
    MoveL Offs(pOrigin,190.93,291.66,0.00),v40,z0,tPen\WObj:=wPaper;
    MoveL Offs(pOrigin,190.22,292.73,0.00),v40,z0,tPen\WObj:=wPaper;
    MoveL Offs(pOrigin,189.44,295.70,0.00),v40,z0,tPen\WObj:=wPaper;
    MoveL Offs(pOrigin,189.23,297.83,0.00),v40,z0,tPen\WObj:=wPaper;
    MoveL Offs(pOrigin,189.65,299.52,0.00),v40,z0,tPen\WObj:=wPaper;
    MoveL Offs(pOrigin,189.65,299.52,0.00),v40,z0,tPen\WObj:=wPaper;
    MoveL Offs(pOrigin,190.43,302.50,0.00),v40,z0,tPen\WObj:=wPaper;
    MoveL Offs(pOrigin,192.13,305.90,0.00),v40,z0,tPen\WObj:=wPaper;
    MoveL Offs(pOrigin,193.19,309.73,0.00),v40,z0,tPen\WObj:=wPaper;
    MoveL Offs(pOrigin,193.97,311.00,0.00),v40,z0,tPen\WObj:=wPaper;
    MoveL Offs(pOrigin,195.39,314.83,0.00),v40,z0,tPen\WObj:=wPaper;
    MoveL Offs(pOrigin,195.39,314.83,0.00),v40,z0,tPen\WObj:=wPaper;
    MoveL Offs(pOrigin,195.95,316.95,0.00),v40,z0,tPen\WObj:=wPaper;
    MoveL Offs(pOrigin,198.36,320.56,0.00),v40,z0,tPen\WObj:=wPaper;
    MoveL Offs(pOrigin,202.82,325.02,0.00),v40,z0,tPen\WObj:=wPaper;
    MoveL Offs(pOrigin,203.25,326.51,0.00),v40,fine,tPen\WObj:=wPaper;
    MoveL Offs(pOrigin,203.25,326.51,6.00),v60,z5,tPen\WObj:=wPaper;
    MoveL Offs(pOrigin,204.52,326.51,6.00),vTravel,z5,tPen\WObj:=wPaper;
    MoveL Offs(pOrigin,204.52,326.51,0.00),v60,z0,tPen\WObj:=wPaper;
    MoveL Offs(pOrigin,203.46,326.58,0.00),v40,z0,tPen\WObj:=wPaper;
    MoveL Offs(pOrigin,203.32,326.94,0.00),v40,z0,tPen\WObj:=wPaper;
    MoveL Offs(pOrigin,204.95,329.49,0.00),v40,z0,tPen\WObj:=wPaper;
    MoveL Offs(pOrigin,208.56,332.89,0.00),v40,z0,tPen\WObj:=wPaper;
    MoveL Offs(pOrigin,213.02,335.08,0.00),v40,z0,tPen\WObj:=wPaper;
    MoveL Offs(pOrigin,218.55,336.50,0.00),v40,z0,tPen\WObj:=wPaper;
    MoveL Offs(pOrigin,227.48,339.69,0.00),v40,z0,tPen\WObj:=wPaper;
    MoveL Offs(pOrigin,230.88,340.33,0.00),v40,z0,tPen\WObj:=wPaper;
    MoveL Offs(pOrigin,235.76,340.33,0.00),v40,z0,tPen\WObj:=wPaper;
    MoveL Offs(pOrigin,237.68,339.90,0.00),v40,z0,tPen\WObj:=wPaper;
    MoveL Offs(pOrigin,241.71,339.69,0.00),v40,z0,tPen\WObj:=wPaper;
    MoveL Offs(pOrigin,241.71,339.05,0.00),v40,z0,tPen\WObj:=wPaper;
    MoveL Offs(pOrigin,241.93,339.62,0.00),v40,z0,tPen\WObj:=wPaper;
    MoveL Offs(pOrigin,242.77,339.90,0.00),v40,z0,tPen\WObj:=wPaper;
    MoveL Offs(pOrigin,252.12,339.69,0.00),v40,z0,tPen\WObj:=wPaper;
    MoveL Offs(pOrigin,255.52,339.05,0.00),v40,z0,tPen\WObj:=wPaper;
    MoveL Offs(pOrigin,258.50,338.06,0.00),v40,z0,tPen\WObj:=wPaper;
    MoveL Offs(pOrigin,259.14,337.56,0.00),v40,fine,tPen\WObj:=wPaper;
    MoveL Offs(pOrigin,259.14,337.56,6.00),v60,z5,tPen\WObj:=wPaper;
    MoveL Offs(pOrigin,259.14,336.29,6.00),vTravel,z5,tPen\WObj:=wPaper;
    MoveL Offs(pOrigin,259.14,336.29,0.00),v60,z0,tPen\WObj:=wPaper;
    MoveL Offs(pOrigin,257.65,336.29,0.00),v40,z0,tPen\WObj:=wPaper;
    MoveL Offs(pOrigin,257.65,336.29,0.00),v40,z0,tPen\WObj:=wPaper;
    MoveL Offs(pOrigin,257.44,335.44,0.00),v40,z0,tPen\WObj:=wPaper;
    MoveL Offs(pOrigin,256.45,334.73,0.00),v40,z0,tPen\WObj:=wPaper;
    MoveL Offs(pOrigin,256.38,333.95,0.00),v40,z0,tPen\WObj:=wPaper;
    MoveL Offs(pOrigin,257.86,331.61,0.00),v40,z0,tPen\WObj:=wPaper;
    MoveL Offs(pOrigin,258.29,328.00,0.00),v40,z0,tPen\WObj:=wPaper;
    MoveL Offs(pOrigin,257.30,324.81,0.00),v40,z0,tPen\WObj:=wPaper;
    MoveL Offs(pOrigin,256.16,324.17,0.00),v40,z0,tPen\WObj:=wPaper;
    MoveL Offs(pOrigin,256.16,324.17,0.00),v40,z0,tPen\WObj:=wPaper;
    MoveL Offs(pOrigin,256.80,326.30,0.00),v40,z0,tPen\WObj:=wPaper;
    MoveL Offs(pOrigin,256.80,327.58,0.00),v40,z0,tPen\WObj:=wPaper;
    MoveL Offs(pOrigin,256.16,330.34,0.00),v40,z0,tPen\WObj:=wPaper;
    MoveL Offs(pOrigin,255.52,330.69,0.00),v40,z0,tPen\WObj:=wPaper;
    MoveL Offs(pOrigin,255.31,330.34,0.00),v40,z0,tPen\WObj:=wPaper;
    MoveL Offs(pOrigin,255.52,326.94,0.00),v40,z0,tPen\WObj:=wPaper;
    MoveL Offs(pOrigin,255.03,325.24,0.00),v40,z0,tPen\WObj:=wPaper;
    MoveL Offs(pOrigin,253.82,323.54,0.00),v40,z0,tPen\WObj:=wPaper;
    MoveL Offs(pOrigin,251.70,322.26,0.00),v40,z0,tPen\WObj:=wPaper;
    MoveL Offs(pOrigin,249.57,320.35,0.00),v40,z0,tPen\WObj:=wPaper;
    MoveL Offs(pOrigin,248.94,319.08,0.00),v40,z0,tPen\WObj:=wPaper;
    MoveL Offs(pOrigin,248.94,319.08,0.00),v40,z0,tPen\WObj:=wPaper;
    MoveL Offs(pOrigin,249.79,318.65,0.00),v40,z0,tPen\WObj:=wPaper;
    MoveL Offs(pOrigin,249.79,318.65,0.00),v40,z0,tPen\WObj:=wPaper;
    MoveL Offs(pOrigin,249.50,317.16,0.00),v40,z0,tPen\WObj:=wPaper;
    MoveL Offs(pOrigin,248.02,315.89,0.00),v40,z0,tPen\WObj:=wPaper;
    MoveL Offs(pOrigin,247.17,313.12,0.00),v40,z0,tPen\WObj:=wPaper;
    MoveL Offs(pOrigin,246.81,312.84,0.00),v40,z0,tPen\WObj:=wPaper;
    MoveL Offs(pOrigin,246.39,313.34,0.00),v40,z0,tPen\WObj:=wPaper;
    MoveL Offs(pOrigin,246.39,314.40,0.00),v40,z0,tPen\WObj:=wPaper;
    MoveL Offs(pOrigin,247.02,317.16,0.00),v40,z0,tPen\WObj:=wPaper;
    MoveL Offs(pOrigin,247.02,317.16,0.00),v40,z0,tPen\WObj:=wPaper;
    MoveL Offs(pOrigin,247.45,318.86,0.00),v40,z0,tPen\WObj:=wPaper;
    MoveL Offs(pOrigin,247.45,318.86,0.00),v40,z0,tPen\WObj:=wPaper;
    MoveL Offs(pOrigin,245.32,318.23,0.00),v40,z0,tPen\WObj:=wPaper;
    MoveL Offs(pOrigin,244.05,318.44,0.00),v40,z0,tPen\WObj:=wPaper;
    MoveL Offs(pOrigin,244.05,318.44,0.00),v40,z0,tPen\WObj:=wPaper;
    MoveL Offs(pOrigin,244.26,319.50,0.00),v40,z0,tPen\WObj:=wPaper;
  ENDPROC

  PROC DrawPart28()
    MoveL Offs(pOrigin,245.11,320.56,0.00),v40,z0,tPen\WObj:=wPaper;
    MoveL Offs(pOrigin,245.11,320.56,0.00),v40,z0,tPen\WObj:=wPaper;
    MoveL Offs(pOrigin,244.26,322.05,0.00),v40,fine,tPen\WObj:=wPaper;
    MoveL Offs(pOrigin,244.26,322.05,6.00),v60,z5,tPen\WObj:=wPaper;
    MoveL Offs(pOrigin,242.77,321.41,6.00),vTravel,z5,tPen\WObj:=wPaper;
    MoveL Offs(pOrigin,242.77,321.41,0.00),v60,z0,tPen\WObj:=wPaper;
    MoveL Offs(pOrigin,241.50,320.99,0.00),v40,z0,tPen\WObj:=wPaper;
    MoveL Offs(pOrigin,239.80,319.29,0.00),v40,z0,tPen\WObj:=wPaper;
    MoveL Offs(pOrigin,238.74,317.59,0.00),v40,z0,tPen\WObj:=wPaper;
    MoveL Offs(pOrigin,238.74,317.59,0.00),v40,z0,tPen\WObj:=wPaper;
    MoveL Offs(pOrigin,237.04,316.95,0.00),v40,z0,tPen\WObj:=wPaper;
    MoveL Offs(pOrigin,237.04,317.38,0.00),v40,z0,tPen\WObj:=wPaper;
    MoveL Offs(pOrigin,235.55,313.76,0.00),v40,z0,tPen\WObj:=wPaper;
    MoveL Offs(pOrigin,235.76,311.85,0.00),v40,z0,tPen\WObj:=wPaper;
    MoveL Offs(pOrigin,235.55,311.42,0.00),v40,z0,tPen\WObj:=wPaper;
    MoveL Offs(pOrigin,235.55,311.42,0.00),v40,z0,tPen\WObj:=wPaper;
    MoveL Offs(pOrigin,235.76,310.79,0.00),v40,z0,tPen\WObj:=wPaper;
    MoveL Offs(pOrigin,237.25,309.51,0.00),v40,fine,tPen\WObj:=wPaper;
    MoveL Offs(pOrigin,237.25,309.51,6.00),v60,z5,tPen\WObj:=wPaper;
    MoveL Offs(pOrigin,238.74,310.15,6.00),vTravel,z5,tPen\WObj:=wPaper;
    MoveL Offs(pOrigin,238.74,310.15,0.00),v60,z0,tPen\WObj:=wPaper;
    MoveL Offs(pOrigin,239.59,310.79,0.00),v40,z0,tPen\WObj:=wPaper;
    MoveL Offs(pOrigin,239.59,311.42,0.00),v40,z0,tPen\WObj:=wPaper;
    MoveL Offs(pOrigin,239.38,313.98,0.00),v40,z0,tPen\WObj:=wPaper;
    MoveL Offs(pOrigin,239.87,315.67,0.00),v40,z0,tPen\WObj:=wPaper;
    MoveL Offs(pOrigin,240.65,316.95,0.00),v40,z0,tPen\WObj:=wPaper;
    MoveL Offs(pOrigin,241.71,317.38,0.00),v40,z0,tPen\WObj:=wPaper;
    MoveL Offs(pOrigin,241.71,317.38,0.00),v40,z0,tPen\WObj:=wPaper;
    MoveL Offs(pOrigin,241.07,315.89,0.00),v40,z0,tPen\WObj:=wPaper;
    MoveL Offs(pOrigin,241.07,312.49,0.00),v40,z0,tPen\WObj:=wPaper;
    MoveL Offs(pOrigin,241.50,311.85,0.00),v40,z0,tPen\WObj:=wPaper;
    MoveL Offs(pOrigin,242.14,311.64,0.00),v40,z0,tPen\WObj:=wPaper;
    MoveL Offs(pOrigin,242.14,311.64,0.00),v40,z0,tPen\WObj:=wPaper;
    MoveL Offs(pOrigin,242.35,314.61,0.00),v40,z0,tPen\WObj:=wPaper;
    MoveL Offs(pOrigin,242.77,315.89,0.00),v40,z0,tPen\WObj:=wPaper;
    MoveL Offs(pOrigin,242.56,317.38,0.00),v40,z0,tPen\WObj:=wPaper;
    MoveL Offs(pOrigin,241.71,317.38,0.00),v40,z0,tPen\WObj:=wPaper;
    MoveL Offs(pOrigin,242.35,317.38,0.00),v40,z0,tPen\WObj:=wPaper;
    MoveL Offs(pOrigin,242.77,318.01,0.00),v40,z0,tPen\WObj:=wPaper;
    MoveL Offs(pOrigin,243.41,318.23,0.00),v40,z0,tPen\WObj:=wPaper;
    MoveL Offs(pOrigin,244.05,318.44,0.00),v40,z0,tPen\WObj:=wPaper;
    MoveL Offs(pOrigin,243.77,318.23,0.00),v40,z0,tPen\WObj:=wPaper;
    MoveL Offs(pOrigin,244.26,316.74,0.00),v40,z0,tPen\WObj:=wPaper;
    MoveL Offs(pOrigin,243.84,315.25,0.00),v40,z0,tPen\WObj:=wPaper;
    MoveL Offs(pOrigin,243.84,313.55,0.00),v40,z0,tPen\WObj:=wPaper;
    MoveL Offs(pOrigin,244.33,312.06,0.00),v40,z0,tPen\WObj:=wPaper;
    MoveL Offs(pOrigin,245.11,311.64,0.00),v40,z0,tPen\WObj:=wPaper;
    MoveL Offs(pOrigin,245.11,311.64,0.00),v40,z0,tPen\WObj:=wPaper;
    MoveL Offs(pOrigin,245.11,314.19,0.00),v40,z0,tPen\WObj:=wPaper;
    MoveL Offs(pOrigin,245.68,315.89,0.00),v40,z0,tPen\WObj:=wPaper;
    MoveL Offs(pOrigin,246.39,316.95,0.00),v40,z0,tPen\WObj:=wPaper;
    MoveL Offs(pOrigin,247.02,317.16,0.00),v40,fine,tPen\WObj:=wPaper;
    MoveL Offs(pOrigin,247.02,317.16,6.00),v60,z5,tPen\WObj:=wPaper;
    MoveL Offs(pOrigin,248.30,316.10,6.00),vTravel,z5,tPen\WObj:=wPaper;
    MoveL Offs(pOrigin,248.30,316.10,0.00),v60,z0,tPen\WObj:=wPaper;
    MoveL Offs(pOrigin,248.73,316.52,0.00),v40,z0,tPen\WObj:=wPaper;
    MoveL Offs(pOrigin,248.30,316.10,0.00),v40,fine,tPen\WObj:=wPaper;
    MoveL Offs(pOrigin,248.30,316.10,6.00),v60,z5,tPen\WObj:=wPaper;
    MoveL Offs(pOrigin,249.36,316.74,6.00),vTravel,z5,tPen\WObj:=wPaper;
    MoveL Offs(pOrigin,249.36,316.74,0.00),v60,z0,tPen\WObj:=wPaper;
    MoveL Offs(pOrigin,248.94,315.04,0.00),v40,z0,tPen\WObj:=wPaper;
    MoveL Offs(pOrigin,248.94,313.12,0.00),v40,z0,tPen\WObj:=wPaper;
    MoveL Offs(pOrigin,249.36,312.70,0.00),v40,fine,tPen\WObj:=wPaper;
    MoveL Offs(pOrigin,249.36,312.70,6.00),v60,z5,tPen\WObj:=wPaper;
    MoveL Offs(pOrigin,249.79,311.21,6.00),vTravel,z5,tPen\WObj:=wPaper;
    MoveL Offs(pOrigin,249.79,311.21,0.00),v60,z0,tPen\WObj:=wPaper;
    MoveL Offs(pOrigin,249.50,312.49,0.00),v40,z0,tPen\WObj:=wPaper;
    MoveL Offs(pOrigin,250.43,315.25,0.00),v40,z0,tPen\WObj:=wPaper;
    MoveL Offs(pOrigin,251.06,315.46,0.00),v40,z0,tPen\WObj:=wPaper;
    MoveL Offs(pOrigin,251.06,315.46,0.00),v40,z0,tPen\WObj:=wPaper;
    MoveL Offs(pOrigin,251.27,316.31,0.00),v40,z0,tPen\WObj:=wPaper;
    MoveL Offs(pOrigin,252.34,317.16,0.00),v40,z0,tPen\WObj:=wPaper;
    MoveL Offs(pOrigin,252.34,317.16,0.00),v40,z0,tPen\WObj:=wPaper;
    MoveL Offs(pOrigin,255.31,318.01,0.00),v40,z0,tPen\WObj:=wPaper;
    MoveL Offs(pOrigin,255.31,318.01,0.00),v40,z0,tPen\WObj:=wPaper;
    MoveL Offs(pOrigin,256.16,318.44,0.00),v40,z0,tPen\WObj:=wPaper;
    MoveL Offs(pOrigin,256.16,318.44,0.00),v40,z0,tPen\WObj:=wPaper;
    MoveL Offs(pOrigin,257.44,318.01,0.00),v40,z0,tPen\WObj:=wPaper;
    MoveL Offs(pOrigin,259.99,319.08,0.00),v40,z0,tPen\WObj:=wPaper;
    MoveL Offs(pOrigin,259.99,319.08,0.00),v40,z0,tPen\WObj:=wPaper;
    MoveL Offs(pOrigin,260.41,319.71,0.00),v40,z0,tPen\WObj:=wPaper;
    MoveL Offs(pOrigin,261.26,319.71,0.00),v40,z0,tPen\WObj:=wPaper;
    MoveL Offs(pOrigin,261.26,319.71,0.00),v40,z0,tPen\WObj:=wPaper;
    MoveL Offs(pOrigin,260.84,318.86,0.00),v40,z0,tPen\WObj:=wPaper;
    MoveL Offs(pOrigin,259.99,319.08,0.00),v40,fine,tPen\WObj:=wPaper;
    MoveL Offs(pOrigin,259.99,319.08,6.00),v60,z5,tPen\WObj:=wPaper;
    MoveL Offs(pOrigin,261.26,319.71,6.00),vTravel,z5,tPen\WObj:=wPaper;
    MoveL Offs(pOrigin,261.26,319.71,0.00),v60,z0,tPen\WObj:=wPaper;
    MoveL Offs(pOrigin,262.33,320.00,0.00),v40,z0,tPen\WObj:=wPaper;
    MoveL Offs(pOrigin,264.45,321.41,0.00),v40,fine,tPen\WObj:=wPaper;
    MoveL Offs(pOrigin,264.45,321.41,6.00),v60,z5,tPen\WObj:=wPaper;
    MoveL Offs(pOrigin,265.51,323.11,6.00),vTravel,z5,tPen\WObj:=wPaper;
    MoveL Offs(pOrigin,265.51,323.11,0.00),v60,z0,tPen\WObj:=wPaper;
    MoveL Offs(pOrigin,266.36,323.96,0.00),v40,z0,tPen\WObj:=wPaper;
    MoveL Offs(pOrigin,265.51,323.11,0.00),v40,fine,tPen\WObj:=wPaper;
    MoveL Offs(pOrigin,265.51,323.11,6.00),v60,z5,tPen\WObj:=wPaper;
    MoveL Offs(pOrigin,264.66,324.60,6.00),vTravel,z5,tPen\WObj:=wPaper;
    MoveL Offs(pOrigin,264.66,324.60,0.00),v60,z0,tPen\WObj:=wPaper;
    MoveL Offs(pOrigin,265.09,325.24,0.00),v40,z0,tPen\WObj:=wPaper;
    MoveL Offs(pOrigin,264.66,324.60,0.00),v40,fine,tPen\WObj:=wPaper;
    MoveL Offs(pOrigin,264.66,324.60,6.00),v60,z5,tPen\WObj:=wPaper;
    MoveL Offs(pOrigin,262.75,323.11,6.00),vTravel,z5,tPen\WObj:=wPaper;
    MoveL Offs(pOrigin,262.75,323.11,0.00),v60,z0,tPen\WObj:=wPaper;
    MoveL Offs(pOrigin,264.02,323.54,0.00),v40,z0,tPen\WObj:=wPaper;
    MoveL Offs(pOrigin,265.37,325.45,0.00),v40,z0,tPen\WObj:=wPaper;
    MoveL Offs(pOrigin,266.15,327.58,0.00),v40,z0,tPen\WObj:=wPaper;
    MoveL Offs(pOrigin,266.36,329.49,0.00),v40,z0,tPen\WObj:=wPaper;
    MoveL Offs(pOrigin,265.73,332.25,0.00),v40,z0,tPen\WObj:=wPaper;
    MoveL Offs(pOrigin,265.09,332.25,0.00),v40,z0,tPen\WObj:=wPaper;
    MoveL Offs(pOrigin,263.39,334.02,0.00),v40,z0,tPen\WObj:=wPaper;
    MoveL Offs(pOrigin,262.11,334.16,0.00),v40,z0,tPen\WObj:=wPaper;
    MoveL Offs(pOrigin,262.11,334.16,0.00),v40,z0,tPen\WObj:=wPaper;
    MoveL Offs(pOrigin,259.21,336.50,0.00),v40,z0,tPen\WObj:=wPaper;
    MoveL Offs(pOrigin,259.21,337.35,0.00),v40,z0,tPen\WObj:=wPaper;
    MoveL Offs(pOrigin,259.77,337.56,0.00),v40,z0,tPen\WObj:=wPaper;
    MoveL Offs(pOrigin,263.60,336.71,0.00),v40,fine,tPen\WObj:=wPaper;
    MoveL Offs(pOrigin,263.60,336.71,6.00),v60,z5,tPen\WObj:=wPaper;
    MoveL Offs(pOrigin,262.11,334.16,6.00),vTravel,z5,tPen\WObj:=wPaper;
    MoveL Offs(pOrigin,262.11,334.16,0.00),v60,z0,tPen\WObj:=wPaper;
    MoveL Offs(pOrigin,262.54,332.67,0.00),v40,z0,tPen\WObj:=wPaper;
  ENDPROC

  PROC DrawPart29()
    MoveL Offs(pOrigin,262.54,332.67,0.00),v40,z0,tPen\WObj:=wPaper;
    MoveL Offs(pOrigin,263.39,332.25,0.00),v40,z0,tPen\WObj:=wPaper;
    MoveL Offs(pOrigin,263.39,331.61,0.00),v40,z0,tPen\WObj:=wPaper;
    MoveL Offs(pOrigin,263.39,331.61,0.00),v40,z0,tPen\WObj:=wPaper;
    MoveL Offs(pOrigin,264.02,330.34,0.00),v40,z0,tPen\WObj:=wPaper;
    MoveL Offs(pOrigin,264.24,327.79,0.00),v40,z0,tPen\WObj:=wPaper;
    MoveL Offs(pOrigin,262.75,323.11,0.00),v40,fine,tPen\WObj:=wPaper;
    MoveL Offs(pOrigin,262.75,323.11,6.00),v60,z5,tPen\WObj:=wPaper;
    MoveL Offs(pOrigin,261.48,321.62,6.00),vTravel,z5,tPen\WObj:=wPaper;
    MoveL Offs(pOrigin,261.48,321.62,0.00),v60,z0,tPen\WObj:=wPaper;
    MoveL Offs(pOrigin,262.33,322.48,0.00),v40,z0,tPen\WObj:=wPaper;
    MoveL Offs(pOrigin,261.48,321.62,0.00),v40,fine,tPen\WObj:=wPaper;
    MoveL Offs(pOrigin,261.48,321.62,6.00),v60,z5,tPen\WObj:=wPaper;
    MoveL Offs(pOrigin,260.41,322.69,6.00),vTravel,z5,tPen\WObj:=wPaper;
    MoveL Offs(pOrigin,260.41,322.69,0.00),v60,z0,tPen\WObj:=wPaper;
    MoveL Offs(pOrigin,260.84,323.11,0.00),v40,z0,tPen\WObj:=wPaper;
    MoveL Offs(pOrigin,260.41,322.69,0.00),v40,fine,tPen\WObj:=wPaper;
    MoveL Offs(pOrigin,260.41,322.69,6.00),v60,z5,tPen\WObj:=wPaper;
    MoveL Offs(pOrigin,259.14,324.17,6.00),vTravel,z5,tPen\WObj:=wPaper;
    MoveL Offs(pOrigin,259.14,324.17,0.00),v60,z0,tPen\WObj:=wPaper;
    MoveL Offs(pOrigin,259.56,324.25,0.00),v40,z0,tPen\WObj:=wPaper;
    MoveL Offs(pOrigin,260.06,325.02,0.00),v40,z0,tPen\WObj:=wPaper;
    MoveL Offs(pOrigin,261.05,328.85,0.00),v40,z0,tPen\WObj:=wPaper;
    MoveL Offs(pOrigin,260.48,331.61,0.00),v40,z0,tPen\WObj:=wPaper;
    MoveL Offs(pOrigin,259.77,332.25,0.00),v40,fine,tPen\WObj:=wPaper;
    MoveL Offs(pOrigin,259.77,332.25,6.00),v60,z5,tPen\WObj:=wPaper;
    MoveL Offs(pOrigin,258.92,334.38,6.00),vTravel,z5,tPen\WObj:=wPaper;
    MoveL Offs(pOrigin,258.92,334.38,0.00),v60,z0,tPen\WObj:=wPaper;
    MoveL Offs(pOrigin,259.14,333.95,0.00),v40,z0,tPen\WObj:=wPaper;
    MoveL Offs(pOrigin,258.92,334.38,0.00),v40,fine,tPen\WObj:=wPaper;
    MoveL Offs(pOrigin,258.92,334.38,6.00),v60,z5,tPen\WObj:=wPaper;
    MoveL Offs(pOrigin,257.65,335.44,6.00),vTravel,z5,tPen\WObj:=wPaper;
    MoveL Offs(pOrigin,257.65,335.44,0.00),v60,z0,tPen\WObj:=wPaper;
    MoveL Offs(pOrigin,258.43,335.01,0.00),v40,z0,tPen\WObj:=wPaper;
    MoveL Offs(pOrigin,259.77,333.10,0.00),v40,z0,tPen\WObj:=wPaper;
    MoveL Offs(pOrigin,259.35,331.40,0.00),v40,z0,tPen\WObj:=wPaper;
    MoveL Offs(pOrigin,259.77,329.70,0.00),v40,z0,tPen\WObj:=wPaper;
    MoveL Offs(pOrigin,259.77,328.00,0.00),v40,z0,tPen\WObj:=wPaper;
    MoveL Offs(pOrigin,258.71,324.81,0.00),v40,z0,tPen\WObj:=wPaper;
    MoveL Offs(pOrigin,259.14,324.17,0.00),v40,z0,tPen\WObj:=wPaper;
    MoveL Offs(pOrigin,259.14,324.17,0.00),v40,z0,tPen\WObj:=wPaper;
    MoveL Offs(pOrigin,259.07,323.33,0.00),v40,z0,tPen\WObj:=wPaper;
    MoveL Offs(pOrigin,257.72,321.62,0.00),v40,z0,tPen\WObj:=wPaper;
    MoveL Offs(pOrigin,257.86,321.13,0.00),v40,z0,tPen\WObj:=wPaper;
    MoveL Offs(pOrigin,258.50,321.27,0.00),v40,z0,tPen\WObj:=wPaper;
    MoveL Offs(pOrigin,260.20,322.69,0.00),v40,z0,tPen\WObj:=wPaper;
    MoveL Offs(pOrigin,262.61,325.88,0.00),v40,z0,tPen\WObj:=wPaper;
    MoveL Offs(pOrigin,263.39,328.85,0.00),v40,z0,tPen\WObj:=wPaper;
    MoveL Offs(pOrigin,262.96,331.61,0.00),v40,z0,tPen\WObj:=wPaper;
    MoveL Offs(pOrigin,262.96,331.61,0.00),v40,z0,tPen\WObj:=wPaper;
    MoveL Offs(pOrigin,262.54,331.83,0.00),v40,z0,tPen\WObj:=wPaper;
    MoveL Offs(pOrigin,262.54,332.67,0.00),v40,fine,tPen\WObj:=wPaper;
    MoveL Offs(pOrigin,262.54,332.67,6.00),v60,z5,tPen\WObj:=wPaper;
    MoveL Offs(pOrigin,266.36,333.52,6.00),vTravel,z5,tPen\WObj:=wPaper;
    MoveL Offs(pOrigin,266.36,333.52,0.00),v60,z0,tPen\WObj:=wPaper;
    MoveL Offs(pOrigin,268.70,333.52,0.00),v40,z0,tPen\WObj:=wPaper;
    MoveL Offs(pOrigin,269.55,333.10,0.00),v40,z0,tPen\WObj:=wPaper;
    MoveL Offs(pOrigin,269.69,332.46,0.00),v40,z0,tPen\WObj:=wPaper;
    MoveL Offs(pOrigin,271.46,330.12,0.00),v40,z0,tPen\WObj:=wPaper;
    MoveL Offs(pOrigin,271.46,330.12,0.00),v40,z0,tPen\WObj:=wPaper;
    MoveL Offs(pOrigin,272.95,329.49,0.00),v40,z0,tPen\WObj:=wPaper;
    MoveL Offs(pOrigin,272.52,328.85,0.00),v40,z0,tPen\WObj:=wPaper;
    MoveL Offs(pOrigin,271.67,329.27,0.00),v40,z0,tPen\WObj:=wPaper;
    MoveL Offs(pOrigin,271.67,329.27,0.00),v40,z0,tPen\WObj:=wPaper;
    MoveL Offs(pOrigin,270.83,328.21,0.00),v40,z0,tPen\WObj:=wPaper;
    MoveL Offs(pOrigin,271.46,327.15,0.00),v40,z0,tPen\WObj:=wPaper;
    MoveL Offs(pOrigin,271.46,327.15,0.00),v40,z0,tPen\WObj:=wPaper;
    MoveL Offs(pOrigin,273.16,327.79,0.00),v40,z0,tPen\WObj:=wPaper;
    MoveL Offs(pOrigin,273.16,327.79,0.00),v40,z0,tPen\WObj:=wPaper;
    MoveL Offs(pOrigin,273.16,328.85,0.00),v40,z0,tPen\WObj:=wPaper;
    MoveL Offs(pOrigin,273.16,328.85,0.00),v40,z0,tPen\WObj:=wPaper;
    MoveL Offs(pOrigin,274.44,329.06,0.00),v40,z0,tPen\WObj:=wPaper;
    MoveL Offs(pOrigin,274.44,329.06,0.00),v40,z0,tPen\WObj:=wPaper;
    MoveL Offs(pOrigin,275.29,328.21,0.00),v40,z0,tPen\WObj:=wPaper;
    MoveL Offs(pOrigin,275.50,328.85,0.00),v40,fine,tPen\WObj:=wPaper;
    MoveL Offs(pOrigin,275.50,328.85,6.00),v60,z5,tPen\WObj:=wPaper;
    MoveL Offs(pOrigin,273.59,330.55,6.00),vTravel,z5,tPen\WObj:=wPaper;
    MoveL Offs(pOrigin,273.59,330.55,0.00),v60,z0,tPen\WObj:=wPaper;
    MoveL Offs(pOrigin,272.95,331.19,0.00),v40,z0,tPen\WObj:=wPaper;
    MoveL Offs(pOrigin,273.59,330.55,0.00),v40,fine,tPen\WObj:=wPaper;
    MoveL Offs(pOrigin,273.59,330.55,6.00),v60,z5,tPen\WObj:=wPaper;
    MoveL Offs(pOrigin,272.52,331.61,6.00),vTravel,z5,tPen\WObj:=wPaper;
    MoveL Offs(pOrigin,272.52,331.61,0.00),v60,z0,tPen\WObj:=wPaper;
    MoveL Offs(pOrigin,272.10,332.04,0.00),v40,z0,tPen\WObj:=wPaper;
    MoveL Offs(pOrigin,272.52,331.61,0.00),v40,fine,tPen\WObj:=wPaper;
    MoveL Offs(pOrigin,272.52,331.61,6.00),v60,z5,tPen\WObj:=wPaper;
    MoveL Offs(pOrigin,270.83,328.42,6.00),vTravel,z5,tPen\WObj:=wPaper;
    MoveL Offs(pOrigin,270.83,328.42,0.00),v60,z0,tPen\WObj:=wPaper;
    MoveL Offs(pOrigin,270.19,327.58,0.00),v40,z0,tPen\WObj:=wPaper;
    MoveL Offs(pOrigin,269.98,326.09,0.00),v40,z0,tPen\WObj:=wPaper;
    MoveL Offs(pOrigin,269.98,326.09,0.00),v40,z0,tPen\WObj:=wPaper;
    MoveL Offs(pOrigin,269.41,324.60,0.00),v40,z0,tPen\WObj:=wPaper;
    MoveL Offs(pOrigin,267.00,320.99,0.00),v40,z0,tPen\WObj:=wPaper;
    MoveL Offs(pOrigin,267.00,320.99,0.00),v40,z0,tPen\WObj:=wPaper;
    MoveL Offs(pOrigin,263.81,319.50,0.00),v40,fine,tPen\WObj:=wPaper;
    MoveL Offs(pOrigin,263.81,319.50,6.00),v60,z5,tPen\WObj:=wPaper;
    MoveL Offs(pOrigin,264.88,318.44,6.00),vTravel,z5,tPen\WObj:=wPaper;
    MoveL Offs(pOrigin,264.88,318.44,0.00),v60,z0,tPen\WObj:=wPaper;
    MoveL Offs(pOrigin,261.05,317.23,0.00),v40,z0,tPen\WObj:=wPaper;
    MoveL Offs(pOrigin,260.20,316.52,0.00),v40,z0,tPen\WObj:=wPaper;
    MoveL Offs(pOrigin,260.20,316.52,0.00),v40,z0,tPen\WObj:=wPaper;
    MoveL Offs(pOrigin,259.77,315.67,0.00),v40,z0,tPen\WObj:=wPaper;
    MoveL Offs(pOrigin,258.08,315.04,0.00),v40,z0,tPen\WObj:=wPaper;
    MoveL Offs(pOrigin,258.08,315.04,0.00),v40,z0,tPen\WObj:=wPaper;
    MoveL Offs(pOrigin,257.79,314.19,0.00),v40,z0,tPen\WObj:=wPaper;
    MoveL Offs(pOrigin,256.66,313.12,0.00),v40,z0,tPen\WObj:=wPaper;
    MoveL Offs(pOrigin,255.81,311.42,0.00),v40,z0,tPen\WObj:=wPaper;
    MoveL Offs(pOrigin,255.74,310.58,0.00),v40,z0,tPen\WObj:=wPaper;
    MoveL Offs(pOrigin,255.74,310.58,0.00),v40,z0,tPen\WObj:=wPaper;
    MoveL Offs(pOrigin,257.23,311.85,0.00),v40,z0,tPen\WObj:=wPaper;
    MoveL Offs(pOrigin,259.77,313.34,0.00),v40,z0,tPen\WObj:=wPaper;
    MoveL Offs(pOrigin,259.77,313.34,0.00),v40,z0,tPen\WObj:=wPaper;
    MoveL Offs(pOrigin,265.94,314.68,0.00),v40,z0,tPen\WObj:=wPaper;
    MoveL Offs(pOrigin,266.15,315.89,0.00),v40,z0,tPen\WObj:=wPaper;
    MoveL Offs(pOrigin,266.15,315.89,0.00),v40,z0,tPen\WObj:=wPaper;
    MoveL Offs(pOrigin,270.61,316.74,0.00),v40,z0,tPen\WObj:=wPaper;
    MoveL Offs(pOrigin,272.10,316.52,0.00),v40,z0,tPen\WObj:=wPaper;
    MoveL Offs(pOrigin,274.23,316.95,0.00),v40,z0,tPen\WObj:=wPaper;
    MoveL Offs(pOrigin,274.65,317.16,0.00),v40,z0,tPen\WObj:=wPaper;
    MoveL Offs(pOrigin,276.14,317.59,0.00),v40,z0,tPen\WObj:=wPaper;
  ENDPROC

  PROC DrawPart30()
    MoveL Offs(pOrigin,276.14,317.59,0.00),v40,z0,tPen\WObj:=wPaper;
    MoveL Offs(pOrigin,277.62,317.87,0.00),v40,z0,tPen\WObj:=wPaper;
    MoveL Offs(pOrigin,279.96,319.43,0.00),v40,z0,tPen\WObj:=wPaper;
    MoveL Offs(pOrigin,281.66,319.71,0.00),v40,z0,tPen\WObj:=wPaper;
    MoveL Offs(pOrigin,281.66,319.71,0.00),v40,z0,tPen\WObj:=wPaper;
    MoveL Offs(pOrigin,282.09,320.35,0.00),v40,z0,tPen\WObj:=wPaper;
    MoveL Offs(pOrigin,283.58,320.35,0.00),v40,z0,tPen\WObj:=wPaper;
    MoveL Offs(pOrigin,283.58,320.56,0.00),v40,fine,tPen\WObj:=wPaper;
    MoveL Offs(pOrigin,283.58,320.56,6.00),v60,z5,tPen\WObj:=wPaper;
    MoveL Offs(pOrigin,284.85,319.29,6.00),vTravel,z5,tPen\WObj:=wPaper;
    MoveL Offs(pOrigin,284.85,319.29,0.00),v60,z0,tPen\WObj:=wPaper;
    MoveL Offs(pOrigin,284.85,320.28,0.00),v40,z0,tPen\WObj:=wPaper;
    MoveL Offs(pOrigin,282.51,321.41,0.00),v40,z0,tPen\WObj:=wPaper;
    MoveL Offs(pOrigin,279.96,321.70,0.00),v40,z0,tPen\WObj:=wPaper;
    MoveL Offs(pOrigin,279.75,322.26,0.00),v40,z0,tPen\WObj:=wPaper;
    MoveL Offs(pOrigin,279.75,322.26,0.00),v40,z0,tPen\WObj:=wPaper;
    MoveL Offs(pOrigin,281.45,322.55,0.00),v40,z0,tPen\WObj:=wPaper;
    MoveL Offs(pOrigin,281.66,323.11,0.00),v40,z0,tPen\WObj:=wPaper;
    MoveL Offs(pOrigin,277.62,324.39,0.00),v40,z0,tPen\WObj:=wPaper;
    MoveL Offs(pOrigin,274.01,323.54,0.00),v40,z0,tPen\WObj:=wPaper;
    MoveL Offs(pOrigin,272.74,323.54,0.00),v40,fine,tPen\WObj:=wPaper;
    MoveL Offs(pOrigin,272.74,323.54,6.00),v60,z5,tPen\WObj:=wPaper;
    MoveL Offs(pOrigin,270.61,326.09,6.00),vTravel,z5,tPen\WObj:=wPaper;
    MoveL Offs(pOrigin,270.61,326.09,0.00),v60,z0,tPen\WObj:=wPaper;
    MoveL Offs(pOrigin,271.46,327.15,0.00),v40,z0,tPen\WObj:=wPaper;
    MoveL Offs(pOrigin,271.04,326.73,0.00),v40,z0,tPen\WObj:=wPaper;
    MoveL Offs(pOrigin,270.19,326.09,0.00),v40,z0,tPen\WObj:=wPaper;
    MoveL Offs(pOrigin,269.98,326.09,0.00),v40,z0,tPen\WObj:=wPaper;
    MoveL Offs(pOrigin,269.55,326.51,0.00),v40,z0,tPen\WObj:=wPaper;
    MoveL Offs(pOrigin,268.27,326.73,0.00),v40,z0,tPen\WObj:=wPaper;
    MoveL Offs(pOrigin,268.27,327.58,0.00),v40,z0,tPen\WObj:=wPaper;
    MoveL Offs(pOrigin,268.91,328.42,0.00),v40,z0,tPen\WObj:=wPaper;
    MoveL Offs(pOrigin,269.12,330.27,0.00),v40,z0,tPen\WObj:=wPaper;
    MoveL Offs(pOrigin,270.83,330.27,0.00),v40,z0,tPen\WObj:=wPaper;
    MoveL Offs(pOrigin,270.40,328.42,0.00),v40,fine,tPen\WObj:=wPaper;
    MoveL Offs(pOrigin,270.40,328.42,6.00),v60,z5,tPen\WObj:=wPaper;
    MoveL Offs(pOrigin,270.61,326.09,6.00),vTravel,z5,tPen\WObj:=wPaper;
    MoveL Offs(pOrigin,270.61,326.09,0.00),v60,z0,tPen\WObj:=wPaper;
    MoveL Offs(pOrigin,271.25,325.45,0.00),v40,z0,tPen\WObj:=wPaper;
    MoveL Offs(pOrigin,275.29,326.73,0.00),v40,z0,tPen\WObj:=wPaper;
    MoveL Offs(pOrigin,277.62,326.73,0.00),v40,z0,tPen\WObj:=wPaper;
    MoveL Offs(pOrigin,279.75,326.09,0.00),v40,fine,tPen\WObj:=wPaper;
    MoveL Offs(pOrigin,279.75,326.09,6.00),v60,z5,tPen\WObj:=wPaper;
    MoveL Offs(pOrigin,279.75,321.62,6.00),vTravel,z5,tPen\WObj:=wPaper;
    MoveL Offs(pOrigin,279.75,321.62,0.00),v60,z0,tPen\WObj:=wPaper;
    MoveL Offs(pOrigin,278.26,320.99,0.00),v40,z0,tPen\WObj:=wPaper;
    MoveL Offs(pOrigin,277.41,320.99,0.00),v40,fine,tPen\WObj:=wPaper;
    MoveL Offs(pOrigin,277.41,320.99,6.00),v60,z5,tPen\WObj:=wPaper;
    MoveL Offs(pOrigin,279.11,319.08,6.00),vTravel,z5,tPen\WObj:=wPaper;
    MoveL Offs(pOrigin,279.11,319.08,0.00),v60,z0,tPen\WObj:=wPaper;
    MoveL Offs(pOrigin,279.54,319.29,0.00),v40,z0,tPen\WObj:=wPaper;
    MoveL Offs(pOrigin,279.11,319.08,0.00),v40,fine,tPen\WObj:=wPaper;
    MoveL Offs(pOrigin,279.11,319.08,6.00),v60,z5,tPen\WObj:=wPaper;
    MoveL Offs(pOrigin,281.66,319.71,6.00),vTravel,z5,tPen\WObj:=wPaper;
    MoveL Offs(pOrigin,281.66,319.71,0.00),v60,z0,tPen\WObj:=wPaper;
    MoveL Offs(pOrigin,284.85,319.29,0.00),v40,z0,tPen\WObj:=wPaper;
    MoveL Offs(pOrigin,284.85,319.29,0.00),v40,z0,tPen\WObj:=wPaper;
    MoveL Offs(pOrigin,286.76,318.01,0.00),v40,z0,tPen\WObj:=wPaper;
    MoveL Offs(pOrigin,286.34,318.23,0.00),v40,z0,tPen\WObj:=wPaper;
    MoveL Offs(pOrigin,287.19,317.80,0.00),v40,z0,tPen\WObj:=wPaper;
    MoveL Offs(pOrigin,288.18,316.74,0.00),v40,z0,tPen\WObj:=wPaper;
    MoveL Offs(pOrigin,288.46,315.46,0.00),v40,z0,tPen\WObj:=wPaper;
    MoveL Offs(pOrigin,288.46,315.46,0.00),v40,z0,tPen\WObj:=wPaper;
    MoveL Offs(pOrigin,286.98,316.10,0.00),v40,z0,tPen\WObj:=wPaper;
    MoveL Offs(pOrigin,286.62,315.89,0.00),v40,z0,tPen\WObj:=wPaper;
    MoveL Offs(pOrigin,287.19,315.11,0.00),v40,z0,tPen\WObj:=wPaper;
    MoveL Offs(pOrigin,288.46,315.04,0.00),v40,fine,tPen\WObj:=wPaper;
    MoveL Offs(pOrigin,288.46,315.04,6.00),v60,z5,tPen\WObj:=wPaper;
    MoveL Offs(pOrigin,288.04,316.74,6.00),vTravel,z5,tPen\WObj:=wPaper;
    MoveL Offs(pOrigin,288.04,316.74,0.00),v60,z0,tPen\WObj:=wPaper;
    MoveL Offs(pOrigin,287.83,317.16,0.00),v40,z0,tPen\WObj:=wPaper;
    MoveL Offs(pOrigin,288.04,316.74,0.00),v40,fine,tPen\WObj:=wPaper;
    MoveL Offs(pOrigin,288.04,316.74,6.00),v60,z5,tPen\WObj:=wPaper;
    MoveL Offs(pOrigin,286.55,316.10,6.00),vTravel,z5,tPen\WObj:=wPaper;
    MoveL Offs(pOrigin,286.55,316.10,0.00),v60,z0,tPen\WObj:=wPaper;
    MoveL Offs(pOrigin,284.42,317.30,0.00),v40,z0,tPen\WObj:=wPaper;
    MoveL Offs(pOrigin,283.36,317.38,0.00),v40,z0,tPen\WObj:=wPaper;
    MoveL Offs(pOrigin,283.36,316.52,0.00),v40,z0,tPen\WObj:=wPaper;
    MoveL Offs(pOrigin,284.85,316.74,0.00),v40,fine,tPen\WObj:=wPaper;
    MoveL Offs(pOrigin,284.85,316.74,6.00),v60,z5,tPen\WObj:=wPaper;
    MoveL Offs(pOrigin,287.19,320.35,6.00),vTravel,z5,tPen\WObj:=wPaper;
    MoveL Offs(pOrigin,287.19,320.35,0.00),v60,z0,tPen\WObj:=wPaper;
    MoveL Offs(pOrigin,286.98,320.77,0.00),v40,z0,tPen\WObj:=wPaper;
    MoveL Offs(pOrigin,287.19,320.35,0.00),v40,fine,tPen\WObj:=wPaper;
    MoveL Offs(pOrigin,287.19,320.35,6.00),v60,z5,tPen\WObj:=wPaper;
    MoveL Offs(pOrigin,286.34,321.41,6.00),vTravel,z5,tPen\WObj:=wPaper;
    MoveL Offs(pOrigin,286.34,321.41,0.00),v60,z0,tPen\WObj:=wPaper;
    MoveL Offs(pOrigin,287.61,320.00,0.00),v40,z0,tPen\WObj:=wPaper;
    MoveL Offs(pOrigin,288.46,319.71,0.00),v40,fine,tPen\WObj:=wPaper;
    MoveL Offs(pOrigin,288.46,319.71,6.00),v60,z5,tPen\WObj:=wPaper;
    MoveL Offs(pOrigin,287.61,322.05,6.00),vTravel,z5,tPen\WObj:=wPaper;
    MoveL Offs(pOrigin,287.61,322.05,0.00),v60,z0,tPen\WObj:=wPaper;
    MoveL Offs(pOrigin,287.19,322.48,0.00),v40,z0,tPen\WObj:=wPaper;
    MoveL Offs(pOrigin,287.61,322.05,0.00),v40,z0,tPen\WObj:=wPaper;
    MoveL Offs(pOrigin,286.98,322.90,0.00),v40,z0,tPen\WObj:=wPaper;
    MoveL Offs(pOrigin,286.34,323.54,0.00),v40,z0,tPen\WObj:=wPaper;
    MoveL Offs(pOrigin,286.98,322.90,0.00),v40,fine,tPen\WObj:=wPaper;
    MoveL Offs(pOrigin,286.98,322.90,6.00),v60,z5,tPen\WObj:=wPaper;
    MoveL Offs(pOrigin,285.91,323.96,6.00),vTravel,z5,tPen\WObj:=wPaper;
    MoveL Offs(pOrigin,285.91,323.96,0.00),v60,z0,tPen\WObj:=wPaper;
    MoveL Offs(pOrigin,285.49,324.39,0.00),v40,z0,tPen\WObj:=wPaper;
    MoveL Offs(pOrigin,285.91,323.96,0.00),v40,fine,tPen\WObj:=wPaper;
    MoveL Offs(pOrigin,285.91,323.96,6.00),v60,z5,tPen\WObj:=wPaper;
    MoveL Offs(pOrigin,285.06,322.69,6.00),vTravel,z5,tPen\WObj:=wPaper;
    MoveL Offs(pOrigin,285.06,322.69,0.00),v60,z0,tPen\WObj:=wPaper;
    MoveL Offs(pOrigin,285.91,321.62,0.00),v40,fine,tPen\WObj:=wPaper;
    MoveL Offs(pOrigin,285.91,321.62,6.00),v60,z5,tPen\WObj:=wPaper;
    MoveL Offs(pOrigin,290.80,316.10,6.00),vTravel,z5,tPen\WObj:=wPaper;
    MoveL Offs(pOrigin,290.80,316.10,0.00),v60,z0,tPen\WObj:=wPaper;
    MoveL Offs(pOrigin,290.38,316.52,0.00),v40,z0,tPen\WObj:=wPaper;
    MoveL Offs(pOrigin,290.80,316.10,0.00),v40,fine,tPen\WObj:=wPaper;
    MoveL Offs(pOrigin,290.80,316.10,6.00),v60,z5,tPen\WObj:=wPaper;
    MoveL Offs(pOrigin,285.70,312.06,6.00),vTravel,z5,tPen\WObj:=wPaper;
    MoveL Offs(pOrigin,285.70,312.06,0.00),v60,z0,tPen\WObj:=wPaper;
    MoveL Offs(pOrigin,282.73,312.27,0.00),v40,z0,tPen\WObj:=wPaper;
    MoveL Offs(pOrigin,282.73,312.27,0.00),v40,z0,tPen\WObj:=wPaper;
    MoveL Offs(pOrigin,281.88,312.49,0.00),v40,z0,tPen\WObj:=wPaper;
    MoveL Offs(pOrigin,279.33,311.85,0.00),v40,z0,tPen\WObj:=wPaper;
    MoveL Offs(pOrigin,278.48,312.06,0.00),v40,fine,tPen\WObj:=wPaper;
    MoveL Offs(pOrigin,278.48,312.06,6.00),v60,z5,tPen\WObj:=wPaper;
  ENDPROC

  PROC DrawPart31()
    MoveL Offs(pOrigin,279.75,309.30,6.00),vTravel,z5,tPen\WObj:=wPaper;
    MoveL Offs(pOrigin,279.75,309.30,0.00),v60,z0,tPen\WObj:=wPaper;
    MoveL Offs(pOrigin,281.02,309.94,0.00),v40,z0,tPen\WObj:=wPaper;
    MoveL Offs(pOrigin,282.73,309.73,0.00),v40,fine,tPen\WObj:=wPaper;
    MoveL Offs(pOrigin,282.73,309.73,6.00),v60,z5,tPen\WObj:=wPaper;
    MoveL Offs(pOrigin,280.81,308.45,6.00),vTravel,z5,tPen\WObj:=wPaper;
    MoveL Offs(pOrigin,280.81,308.45,0.00),v60,z0,tPen\WObj:=wPaper;
    MoveL Offs(pOrigin,280.17,307.60,0.00),v40,z0,tPen\WObj:=wPaper;
    MoveL Offs(pOrigin,280.81,308.45,0.00),v40,z0,tPen\WObj:=wPaper;
    MoveL Offs(pOrigin,284.85,308.02,0.00),v40,z0,tPen\WObj:=wPaper;
    MoveL Offs(pOrigin,286.76,306.96,0.00),v40,fine,tPen\WObj:=wPaper;
    MoveL Offs(pOrigin,286.76,306.96,6.00),v60,z5,tPen\WObj:=wPaper;
    MoveL Offs(pOrigin,285.06,304.41,6.00),vTravel,z5,tPen\WObj:=wPaper;
    MoveL Offs(pOrigin,285.06,304.41,0.00),v60,z0,tPen\WObj:=wPaper;
    MoveL Offs(pOrigin,284.00,303.42,0.00),v40,z0,tPen\WObj:=wPaper;
    MoveL Offs(pOrigin,283.08,304.55,0.00),v40,z0,tPen\WObj:=wPaper;
    MoveL Offs(pOrigin,280.60,305.69,0.00),v40,z0,tPen\WObj:=wPaper;
    MoveL Offs(pOrigin,280.60,306.25,0.00),v40,z0,tPen\WObj:=wPaper;
    MoveL Offs(pOrigin,281.45,306.54,0.00),v40,z0,tPen\WObj:=wPaper;
    MoveL Offs(pOrigin,280.39,306.33,0.00),v40,z0,tPen\WObj:=wPaper;
    MoveL Offs(pOrigin,279.11,306.33,0.00),v40,z0,tPen\WObj:=wPaper;
    MoveL Offs(pOrigin,278.69,306.75,0.00),v40,z0,tPen\WObj:=wPaper;
    MoveL Offs(pOrigin,278.69,306.75,0.00),v40,z0,tPen\WObj:=wPaper;
    MoveL Offs(pOrigin,275.08,306.96,0.00),v40,fine,tPen\WObj:=wPaper;
    MoveL Offs(pOrigin,275.08,306.96,6.00),v60,z5,tPen\WObj:=wPaper;
    MoveL Offs(pOrigin,273.59,305.69,6.00),vTravel,z5,tPen\WObj:=wPaper;
    MoveL Offs(pOrigin,273.59,305.69,0.00),v60,z0,tPen\WObj:=wPaper;
    MoveL Offs(pOrigin,270.40,306.75,0.00),v40,z0,tPen\WObj:=wPaper;
    MoveL Offs(pOrigin,270.40,306.75,0.00),v40,z0,tPen\WObj:=wPaper;
    MoveL Offs(pOrigin,269.34,307.81,0.00),v40,z0,tPen\WObj:=wPaper;
    MoveL Offs(pOrigin,268.70,307.39,0.00),v40,z0,tPen\WObj:=wPaper;
    MoveL Offs(pOrigin,268.70,307.39,0.00),v40,z0,tPen\WObj:=wPaper;
    MoveL Offs(pOrigin,265.30,307.60,0.00),v40,z0,tPen\WObj:=wPaper;
    MoveL Offs(pOrigin,264.95,307.81,0.00),v40,z0,tPen\WObj:=wPaper;
    MoveL Offs(pOrigin,264.88,308.66,0.00),v40,z0,tPen\WObj:=wPaper;
    MoveL Offs(pOrigin,264.88,308.66,0.00),v40,z0,tPen\WObj:=wPaper;
    MoveL Offs(pOrigin,265.94,309.30,0.00),v40,z0,tPen\WObj:=wPaper;
    MoveL Offs(pOrigin,265.94,309.30,0.00),v40,z0,tPen\WObj:=wPaper;
    MoveL Offs(pOrigin,267.00,308.66,0.00),v40,z0,tPen\WObj:=wPaper;
    MoveL Offs(pOrigin,268.49,308.59,0.00),v40,z0,tPen\WObj:=wPaper;
    MoveL Offs(pOrigin,269.34,308.02,0.00),v40,z0,tPen\WObj:=wPaper;
    MoveL Offs(pOrigin,272.74,307.60,0.00),v40,fine,tPen\WObj:=wPaper;
    MoveL Offs(pOrigin,272.74,307.60,6.00),v60,z5,tPen\WObj:=wPaper;
    MoveL Offs(pOrigin,273.16,309.73,6.00),vTravel,z5,tPen\WObj:=wPaper;
    MoveL Offs(pOrigin,273.16,309.73,0.00),v60,z0,tPen\WObj:=wPaper;
    MoveL Offs(pOrigin,272.52,310.15,0.00),v40,z0,tPen\WObj:=wPaper;
    MoveL Offs(pOrigin,268.49,310.58,0.00),v40,z0,tPen\WObj:=wPaper;
    MoveL Offs(pOrigin,266.58,310.22,0.00),v40,z0,tPen\WObj:=wPaper;
    MoveL Offs(pOrigin,265.94,309.73,0.00),v40,z0,tPen\WObj:=wPaper;
    MoveL Offs(pOrigin,265.94,309.73,0.00),v40,z0,tPen\WObj:=wPaper;
    MoveL Offs(pOrigin,265.09,310.29,0.00),v40,z0,tPen\WObj:=wPaper;
    MoveL Offs(pOrigin,261.05,309.30,0.00),v40,z0,tPen\WObj:=wPaper;
    MoveL Offs(pOrigin,260.20,308.88,0.00),v40,z0,tPen\WObj:=wPaper;
    MoveL Offs(pOrigin,261.69,310.65,0.00),v40,z0,tPen\WObj:=wPaper;
    MoveL Offs(pOrigin,263.60,311.64,0.00),v40,z0,tPen\WObj:=wPaper;
    MoveL Offs(pOrigin,263.60,311.64,0.00),v40,z0,tPen\WObj:=wPaper;
    MoveL Offs(pOrigin,264.24,311.64,0.00),v40,z0,tPen\WObj:=wPaper;
    MoveL Offs(pOrigin,264.66,312.27,0.00),v40,z0,tPen\WObj:=wPaper;
    MoveL Offs(pOrigin,264.66,312.27,0.00),v40,z0,tPen\WObj:=wPaper;
    MoveL Offs(pOrigin,266.79,312.27,0.00),v40,z0,tPen\WObj:=wPaper;
    MoveL Offs(pOrigin,267.21,312.91,0.00),v40,z0,tPen\WObj:=wPaper;
    MoveL Offs(pOrigin,267.21,312.91,0.00),v40,z0,tPen\WObj:=wPaper;
    MoveL Offs(pOrigin,267.00,313.34,0.00),v40,z0,tPen\WObj:=wPaper;
    MoveL Offs(pOrigin,267.21,313.76,0.00),v40,z0,tPen\WObj:=wPaper;
    MoveL Offs(pOrigin,268.06,314.40,0.00),v40,z0,tPen\WObj:=wPaper;
    MoveL Offs(pOrigin,267.64,314.40,0.00),v40,z0,tPen\WObj:=wPaper;
    MoveL Offs(pOrigin,266.15,314.61,0.00),v40,fine,tPen\WObj:=wPaper;
    MoveL Offs(pOrigin,266.15,314.61,6.00),v60,z5,tPen\WObj:=wPaper;
    MoveL Offs(pOrigin,268.27,313.98,6.00),vTravel,z5,tPen\WObj:=wPaper;
    MoveL Offs(pOrigin,268.27,313.98,0.00),v60,z0,tPen\WObj:=wPaper;
    MoveL Offs(pOrigin,268.20,312.91,0.00),v40,z0,tPen\WObj:=wPaper;
    MoveL Offs(pOrigin,268.49,312.70,0.00),v40,z0,tPen\WObj:=wPaper;
    MoveL Offs(pOrigin,269.12,312.77,0.00),v40,z0,tPen\WObj:=wPaper;
    MoveL Offs(pOrigin,270.61,313.76,0.00),v40,z0,tPen\WObj:=wPaper;
    MoveL Offs(pOrigin,269.76,313.55,0.00),v40,z0,tPen\WObj:=wPaper;
    MoveL Offs(pOrigin,269.34,313.98,0.00),v40,z0,tPen\WObj:=wPaper;
    MoveL Offs(pOrigin,268.27,313.98,0.00),v40,fine,tPen\WObj:=wPaper;
    MoveL Offs(pOrigin,268.27,313.98,6.00),v60,z5,tPen\WObj:=wPaper;
    MoveL Offs(pOrigin,269.12,312.91,6.00),vTravel,z5,tPen\WObj:=wPaper;
    MoveL Offs(pOrigin,269.12,312.91,0.00),v60,z0,tPen\WObj:=wPaper;
    MoveL Offs(pOrigin,269.76,313.55,0.00),v40,fine,tPen\WObj:=wPaper;
    MoveL Offs(pOrigin,269.76,313.55,6.00),v60,z5,tPen\WObj:=wPaper;
    MoveL Offs(pOrigin,268.27,310.36,6.00),vTravel,z5,tPen\WObj:=wPaper;
    MoveL Offs(pOrigin,268.27,310.36,0.00),v60,z0,tPen\WObj:=wPaper;
    MoveL Offs(pOrigin,268.91,309.73,0.00),v40,z0,tPen\WObj:=wPaper;
    MoveL Offs(pOrigin,270.12,310.01,0.00),v40,z0,tPen\WObj:=wPaper;
    MoveL Offs(pOrigin,270.83,309.51,0.00),v40,z0,tPen\WObj:=wPaper;
    MoveL Offs(pOrigin,271.82,309.80,0.00),v40,z0,tPen\WObj:=wPaper;
    MoveL Offs(pOrigin,272.52,309.30,0.00),v40,z0,tPen\WObj:=wPaper;
    MoveL Offs(pOrigin,274.01,309.73,0.00),v40,fine,tPen\WObj:=wPaper;
    MoveL Offs(pOrigin,274.01,309.73,6.00),v60,z5,tPen\WObj:=wPaper;
    MoveL Offs(pOrigin,270.40,306.75,6.00),vTravel,z5,tPen\WObj:=wPaper;
    MoveL Offs(pOrigin,270.40,306.75,0.00),v60,z0,tPen\WObj:=wPaper;
    MoveL Offs(pOrigin,269.98,305.97,0.00),v40,z0,tPen\WObj:=wPaper;
    MoveL Offs(pOrigin,269.12,305.97,0.00),v40,z0,tPen\WObj:=wPaper;
    MoveL Offs(pOrigin,268.70,307.39,0.00),v40,fine,tPen\WObj:=wPaper;
    MoveL Offs(pOrigin,268.70,307.39,6.00),v60,z5,tPen\WObj:=wPaper;
    MoveL Offs(pOrigin,270.19,305.90,6.00),vTravel,z5,tPen\WObj:=wPaper;
    MoveL Offs(pOrigin,270.19,305.90,0.00),v60,z0,tPen\WObj:=wPaper;
    MoveL Offs(pOrigin,270.61,305.26,0.00),v40,z0,tPen\WObj:=wPaper;
    MoveL Offs(pOrigin,271.89,305.05,0.00),v40,z0,tPen\WObj:=wPaper;
    MoveL Offs(pOrigin,272.31,304.62,0.00),v40,z0,tPen\WObj:=wPaper;
    MoveL Offs(pOrigin,272.31,304.62,0.00),v40,z0,tPen\WObj:=wPaper;
    MoveL Offs(pOrigin,274.01,305.33,0.00),v40,z0,tPen\WObj:=wPaper;
    MoveL Offs(pOrigin,276.56,304.41,0.00),v40,z0,tPen\WObj:=wPaper;
    MoveL Offs(pOrigin,276.56,304.41,0.00),v40,z0,tPen\WObj:=wPaper;
    MoveL Offs(pOrigin,276.77,302.71,0.00),v40,z0,tPen\WObj:=wPaper;
    MoveL Offs(pOrigin,276.77,302.71,0.00),v40,z0,tPen\WObj:=wPaper;
    MoveL Offs(pOrigin,278.69,301.37,0.00),v40,z0,tPen\WObj:=wPaper;
    MoveL Offs(pOrigin,279.96,300.94,0.00),v40,z0,tPen\WObj:=wPaper;
    MoveL Offs(pOrigin,280.60,300.16,0.00),v40,fine,tPen\WObj:=wPaper;
    MoveL Offs(pOrigin,280.60,300.16,6.00),v60,z5,tPen\WObj:=wPaper;
    MoveL Offs(pOrigin,281.24,302.29,6.00),vTravel,z5,tPen\WObj:=wPaper;
    MoveL Offs(pOrigin,281.24,302.29,0.00),v60,z0,tPen\WObj:=wPaper;
    MoveL Offs(pOrigin,282.30,302.71,0.00),v40,z0,tPen\WObj:=wPaper;
    MoveL Offs(pOrigin,283.08,302.43,0.00),v40,z0,tPen\WObj:=wPaper;
    MoveL Offs(pOrigin,283.58,301.08,0.00),v40,z0,tPen\WObj:=wPaper;
    MoveL Offs(pOrigin,285.27,301.08,0.00),v40,z0,tPen\WObj:=wPaper;
    MoveL Offs(pOrigin,285.49,301.44,0.00),v40,z0,tPen\WObj:=wPaper;
    MoveL Offs(pOrigin,285.13,302.50,0.00),v40,z0,tPen\WObj:=wPaper;
  ENDPROC

  PROC DrawPart32()
    MoveL Offs(pOrigin,284.42,303.35,0.00),v40,z0,tPen\WObj:=wPaper;
    MoveL Offs(pOrigin,283.36,303.77,0.00),v40,z0,tPen\WObj:=wPaper;
    MoveL Offs(pOrigin,281.45,303.99,0.00),v40,z0,tPen\WObj:=wPaper;
    MoveL Offs(pOrigin,280.81,303.56,0.00),v40,z0,tPen\WObj:=wPaper;
    MoveL Offs(pOrigin,280.81,303.56,0.00),v40,z0,tPen\WObj:=wPaper;
    MoveL Offs(pOrigin,280.81,302.50,0.00),v40,z0,tPen\WObj:=wPaper;
    MoveL Offs(pOrigin,281.24,302.29,0.00),v40,z0,tPen\WObj:=wPaper;
    MoveL Offs(pOrigin,281.24,302.29,0.00),v40,z0,tPen\WObj:=wPaper;
    MoveL Offs(pOrigin,281.24,300.45,0.00),v40,z0,tPen\WObj:=wPaper;
    MoveL Offs(pOrigin,283.36,301.01,0.00),v40,fine,tPen\WObj:=wPaper;
    MoveL Offs(pOrigin,283.36,301.01,6.00),v60,z5,tPen\WObj:=wPaper;
    MoveL Offs(pOrigin,285.49,301.01,6.00),vTravel,z5,tPen\WObj:=wPaper;
    MoveL Offs(pOrigin,285.49,301.01,0.00),v60,z0,tPen\WObj:=wPaper;
    MoveL Offs(pOrigin,285.91,301.01,0.00),v40,z0,tPen\WObj:=wPaper;
    MoveL Offs(pOrigin,286.55,300.38,0.00),v40,z0,tPen\WObj:=wPaper;
    MoveL Offs(pOrigin,286.55,299.95,0.00),v40,fine,tPen\WObj:=wPaper;
    MoveL Offs(pOrigin,286.55,299.95,6.00),v60,z5,tPen\WObj:=wPaper;
    MoveL Offs(pOrigin,288.25,301.44,6.00),vTravel,z5,tPen\WObj:=wPaper;
    MoveL Offs(pOrigin,288.25,301.44,0.00),v60,z0,tPen\WObj:=wPaper;
    MoveL Offs(pOrigin,288.04,301.86,0.00),v40,z0,tPen\WObj:=wPaper;
    MoveL Offs(pOrigin,288.25,301.44,0.00),v40,z0,tPen\WObj:=wPaper;
    MoveL Offs(pOrigin,288.67,301.23,0.00),v40,z0,tPen\WObj:=wPaper;
    MoveL Offs(pOrigin,288.89,300.80,0.00),v40,z0,tPen\WObj:=wPaper;
    MoveL Offs(pOrigin,288.67,301.23,0.00),v40,fine,tPen\WObj:=wPaper;
    MoveL Offs(pOrigin,288.67,301.23,6.00),v60,z5,tPen\WObj:=wPaper;
    MoveL Offs(pOrigin,290.38,302.92,6.00),vTravel,z5,tPen\WObj:=wPaper;
    MoveL Offs(pOrigin,290.38,302.92,0.00),v60,z0,tPen\WObj:=wPaper;
    MoveL Offs(pOrigin,290.23,302.29,0.00),v40,z0,tPen\WObj:=wPaper;
    MoveL Offs(pOrigin,290.59,301.72,0.00),v40,z0,tPen\WObj:=wPaper;
    MoveL Offs(pOrigin,292.71,301.01,0.00),v40,z0,tPen\WObj:=wPaper;
    MoveL Offs(pOrigin,292.71,301.01,0.00),v40,z0,tPen\WObj:=wPaper;
    MoveL Offs(pOrigin,293.14,300.59,0.00),v40,z0,tPen\WObj:=wPaper;
    MoveL Offs(pOrigin,294.20,300.59,0.00),v40,z0,tPen\WObj:=wPaper;
    MoveL Offs(pOrigin,295.26,301.86,0.00),v40,z0,tPen\WObj:=wPaper;
    MoveL Offs(pOrigin,294.84,301.65,0.00),v40,z0,tPen\WObj:=wPaper;
    MoveL Offs(pOrigin,295.26,301.86,0.00),v40,z0,tPen\WObj:=wPaper;
    MoveL Offs(pOrigin,294.84,301.65,0.00),v40,z0,tPen\WObj:=wPaper;
    MoveL Offs(pOrigin,294.41,301.01,0.00),v40,z0,tPen\WObj:=wPaper;
    MoveL Offs(pOrigin,293.99,301.44,0.00),v40,z0,tPen\WObj:=wPaper;
    MoveL Offs(pOrigin,293.14,301.44,0.00),v40,z0,tPen\WObj:=wPaper;
    MoveL Offs(pOrigin,292.71,301.01,0.00),v40,fine,tPen\WObj:=wPaper;
    MoveL Offs(pOrigin,292.71,301.01,6.00),v60,z5,tPen\WObj:=wPaper;
    MoveL Offs(pOrigin,291.23,298.04,6.00),vTravel,z5,tPen\WObj:=wPaper;
    MoveL Offs(pOrigin,291.23,298.04,0.00),v60,z0,tPen\WObj:=wPaper;
    MoveL Offs(pOrigin,293.99,297.61,0.00),v40,z0,tPen\WObj:=wPaper;
    MoveL Offs(pOrigin,293.99,297.61,0.00),v40,z0,tPen\WObj:=wPaper;
    MoveL Offs(pOrigin,293.56,296.83,0.00),v40,z0,tPen\WObj:=wPaper;
    MoveL Offs(pOrigin,292.08,296.76,0.00),v40,z0,tPen\WObj:=wPaper;
    MoveL Offs(pOrigin,291.23,297.61,0.00),v40,fine,tPen\WObj:=wPaper;
    MoveL Offs(pOrigin,291.23,297.61,6.00),v60,z5,tPen\WObj:=wPaper;
    MoveL Offs(pOrigin,288.67,296.76,6.00),vTravel,z5,tPen\WObj:=wPaper;
    MoveL Offs(pOrigin,288.67,296.76,0.00),v60,z0,tPen\WObj:=wPaper;
    MoveL Offs(pOrigin,288.04,297.40,0.00),v40,z0,tPen\WObj:=wPaper;
    MoveL Offs(pOrigin,288.67,296.76,0.00),v40,fine,tPen\WObj:=wPaper;
    MoveL Offs(pOrigin,288.67,296.76,6.00),v60,z5,tPen\WObj:=wPaper;
    MoveL Offs(pOrigin,284.42,299.10,6.00),vTravel,z5,tPen\WObj:=wPaper;
    MoveL Offs(pOrigin,284.42,299.10,0.00),v60,z0,tPen\WObj:=wPaper;
    MoveL Offs(pOrigin,284.21,299.52,0.00),v40,z0,tPen\WObj:=wPaper;
    MoveL Offs(pOrigin,284.42,299.10,0.00),v40,fine,tPen\WObj:=wPaper;
    MoveL Offs(pOrigin,284.42,299.10,6.00),v60,z5,tPen\WObj:=wPaper;
    MoveL Offs(pOrigin,280.39,295.27,6.00),vTravel,z5,tPen\WObj:=wPaper;
    MoveL Offs(pOrigin,280.39,295.27,0.00),v60,z0,tPen\WObj:=wPaper;
    MoveL Offs(pOrigin,280.60,294.42,0.00),v40,z0,tPen\WObj:=wPaper;
    MoveL Offs(pOrigin,281.66,293.79,0.00),v40,fine,tPen\WObj:=wPaper;
    MoveL Offs(pOrigin,281.66,293.79,6.00),v60,z5,tPen\WObj:=wPaper;
    MoveL Offs(pOrigin,278.48,294.21,6.00),vTravel,z5,tPen\WObj:=wPaper;
    MoveL Offs(pOrigin,278.48,294.21,0.00),v60,z0,tPen\WObj:=wPaper;
    MoveL Offs(pOrigin,279.18,292.30,0.00),v40,z0,tPen\WObj:=wPaper;
    MoveL Offs(pOrigin,280.10,291.02,0.00),v40,z0,tPen\WObj:=wPaper;
    MoveL Offs(pOrigin,280.39,289.33,0.00),v40,z0,tPen\WObj:=wPaper;
    MoveL Offs(pOrigin,280.39,289.33,0.00),v40,z0,tPen\WObj:=wPaper;
    MoveL Offs(pOrigin,282.51,288.33,0.00),v40,z0,tPen\WObj:=wPaper;
    MoveL Offs(pOrigin,283.58,287.20,0.00),v40,fine,tPen\WObj:=wPaper;
    MoveL Offs(pOrigin,283.58,287.20,6.00),v60,z5,tPen\WObj:=wPaper;
    MoveL Offs(pOrigin,284.85,284.65,6.00),vTravel,z5,tPen\WObj:=wPaper;
    MoveL Offs(pOrigin,284.85,284.65,0.00),v60,z0,tPen\WObj:=wPaper;
    MoveL Offs(pOrigin,286.34,284.44,0.00),v40,fine,tPen\WObj:=wPaper;
    MoveL Offs(pOrigin,286.34,284.44,6.00),v60,z5,tPen\WObj:=wPaper;
    MoveL Offs(pOrigin,279.96,285.92,6.00),vTravel,z5,tPen\WObj:=wPaper;
    MoveL Offs(pOrigin,279.96,285.92,0.00),v60,z0,tPen\WObj:=wPaper;
    MoveL Offs(pOrigin,279.75,288.05,0.00),v40,z0,tPen\WObj:=wPaper;
    MoveL Offs(pOrigin,280.39,289.33,0.00),v40,fine,tPen\WObj:=wPaper;
    MoveL Offs(pOrigin,280.39,289.33,6.00),v60,z5,tPen\WObj:=wPaper;
    MoveL Offs(pOrigin,278.48,294.21,6.00),vTravel,z5,tPen\WObj:=wPaper;
    MoveL Offs(pOrigin,278.48,294.21,0.00),v60,z0,tPen\WObj:=wPaper;
    MoveL Offs(pOrigin,278.69,295.70,0.00),v40,fine,tPen\WObj:=wPaper;
    MoveL Offs(pOrigin,278.69,295.70,6.00),v60,z5,tPen\WObj:=wPaper;
    MoveL Offs(pOrigin,277.62,298.89,6.00),vTravel,z5,tPen\WObj:=wPaper;
    MoveL Offs(pOrigin,277.62,298.89,0.00),v60,z0,tPen\WObj:=wPaper;
    MoveL Offs(pOrigin,276.56,299.52,0.00),v40,z0,tPen\WObj:=wPaper;
    MoveL Offs(pOrigin,275.43,301.86,0.00),v40,z0,tPen\WObj:=wPaper;
    MoveL Offs(pOrigin,275.92,302.64,0.00),v40,z0,tPen\WObj:=wPaper;
    MoveL Offs(pOrigin,276.77,302.71,0.00),v40,fine,tPen\WObj:=wPaper;
    MoveL Offs(pOrigin,276.77,302.71,6.00),v60,z5,tPen\WObj:=wPaper;
    MoveL Offs(pOrigin,275.29,302.29,6.00),vTravel,z5,tPen\WObj:=wPaper;
    MoveL Offs(pOrigin,275.29,302.29,0.00),v60,z0,tPen\WObj:=wPaper;
    MoveL Offs(pOrigin,274.65,302.36,0.00),v40,z0,tPen\WObj:=wPaper;
    MoveL Offs(pOrigin,273.80,303.49,0.00),v40,z0,tPen\WObj:=wPaper;
    MoveL Offs(pOrigin,272.31,303.99,0.00),v40,fine,tPen\WObj:=wPaper;
    MoveL Offs(pOrigin,272.31,303.99,6.00),v60,z5,tPen\WObj:=wPaper;
    MoveL Offs(pOrigin,276.56,304.41,6.00),vTravel,z5,tPen\WObj:=wPaper;
    MoveL Offs(pOrigin,276.56,304.41,0.00),v60,z0,tPen\WObj:=wPaper;
    MoveL Offs(pOrigin,277.62,304.62,0.00),v40,z0,tPen\WObj:=wPaper;
    MoveL Offs(pOrigin,278.90,304.41,0.00),v40,z0,tPen\WObj:=wPaper;
    MoveL Offs(pOrigin,280.81,303.56,0.00),v40,fine,tPen\WObj:=wPaper;
    MoveL Offs(pOrigin,280.81,303.56,6.00),v60,z5,tPen\WObj:=wPaper;
    MoveL Offs(pOrigin,278.69,307.60,6.00),vTravel,z5,tPen\WObj:=wPaper;
    MoveL Offs(pOrigin,278.69,307.60,0.00),v60,z0,tPen\WObj:=wPaper;
    MoveL Offs(pOrigin,278.48,308.88,0.00),v40,z0,tPen\WObj:=wPaper;
    MoveL Offs(pOrigin,279.75,309.30,0.00),v40,z0,tPen\WObj:=wPaper;
    MoveL Offs(pOrigin,279.75,309.30,0.00),v40,z0,tPen\WObj:=wPaper;
    MoveL Offs(pOrigin,280.17,308.66,0.00),v40,z0,tPen\WObj:=wPaper;
    MoveL Offs(pOrigin,280.81,308.45,0.00),v40,fine,tPen\WObj:=wPaper;
    MoveL Offs(pOrigin,280.81,308.45,6.00),v60,z5,tPen\WObj:=wPaper;
    MoveL Offs(pOrigin,274.01,315.25,6.00),vTravel,z5,tPen\WObj:=wPaper;
    MoveL Offs(pOrigin,274.01,315.25,0.00),v60,z0,tPen\WObj:=wPaper;
    MoveL Offs(pOrigin,274.23,315.67,0.00),v40,z0,tPen\WObj:=wPaper;
    MoveL Offs(pOrigin,274.01,315.25,0.00),v40,fine,tPen\WObj:=wPaper;
    MoveL Offs(pOrigin,274.01,315.25,6.00),v60,z5,tPen\WObj:=wPaper;
    MoveL Offs(pOrigin,271.89,319.50,6.00),vTravel,z5,tPen\WObj:=wPaper;
  ENDPROC

  PROC DrawPart33()
    MoveL Offs(pOrigin,271.89,319.50,0.00),v60,z0,tPen\WObj:=wPaper;
    MoveL Offs(pOrigin,270.40,318.86,0.00),v40,z0,tPen\WObj:=wPaper;
    MoveL Offs(pOrigin,268.91,318.86,0.00),v40,z0,tPen\WObj:=wPaper;
    MoveL Offs(pOrigin,267.21,318.23,0.00),v40,z0,tPen\WObj:=wPaper;
    MoveL Offs(pOrigin,266.36,318.44,0.00),v40,z0,tPen\WObj:=wPaper;
    MoveL Offs(pOrigin,264.88,317.80,0.00),v40,z0,tPen\WObj:=wPaper;
    MoveL Offs(pOrigin,264.88,317.80,0.00),v40,z0,tPen\WObj:=wPaper;
    MoveL Offs(pOrigin,264.02,317.59,0.00),v40,z0,tPen\WObj:=wPaper;
    MoveL Offs(pOrigin,263.81,317.80,0.00),v40,fine,tPen\WObj:=wPaper;
    MoveL Offs(pOrigin,263.81,317.80,6.00),v60,z5,tPen\WObj:=wPaper;
    MoveL Offs(pOrigin,264.88,318.44,6.00),vTravel,z5,tPen\WObj:=wPaper;
    MoveL Offs(pOrigin,264.88,318.44,0.00),v60,z0,tPen\WObj:=wPaper;
    MoveL Offs(pOrigin,265.73,318.65,0.00),v40,z0,tPen\WObj:=wPaper;
    MoveL Offs(pOrigin,265.94,318.44,0.00),v40,fine,tPen\WObj:=wPaper;
    MoveL Offs(pOrigin,265.94,318.44,6.00),v60,z5,tPen\WObj:=wPaper;
    MoveL Offs(pOrigin,268.49,318.86,6.00),vTravel,z5,tPen\WObj:=wPaper;
    MoveL Offs(pOrigin,268.49,318.86,0.00),v60,z0,tPen\WObj:=wPaper;
    MoveL Offs(pOrigin,268.70,320.35,0.00),v40,z0,tPen\WObj:=wPaper;
    MoveL Offs(pOrigin,268.49,320.35,0.00),v40,fine,tPen\WObj:=wPaper;
    MoveL Offs(pOrigin,268.49,320.35,6.00),v60,z5,tPen\WObj:=wPaper;
    MoveL Offs(pOrigin,262.11,317.38,6.00),vTravel,z5,tPen\WObj:=wPaper;
    MoveL Offs(pOrigin,262.11,317.38,0.00),v60,z0,tPen\WObj:=wPaper;
    MoveL Offs(pOrigin,262.11,316.31,0.00),v40,z0,tPen\WObj:=wPaper;
    MoveL Offs(pOrigin,262.11,316.31,0.00),v40,z0,tPen\WObj:=wPaper;
    MoveL Offs(pOrigin,260.84,316.10,0.00),v40,z0,tPen\WObj:=wPaper;
    MoveL Offs(pOrigin,260.62,316.52,0.00),v40,fine,tPen\WObj:=wPaper;
    MoveL Offs(pOrigin,260.62,316.52,6.00),v60,z5,tPen\WObj:=wPaper;
    MoveL Offs(pOrigin,258.71,315.25,6.00),vTravel,z5,tPen\WObj:=wPaper;
    MoveL Offs(pOrigin,258.71,315.25,0.00),v60,z0,tPen\WObj:=wPaper;
    MoveL Offs(pOrigin,259.14,315.46,0.00),v40,z0,tPen\WObj:=wPaper;
    MoveL Offs(pOrigin,258.71,315.25,0.00),v40,z0,tPen\WObj:=wPaper;
    MoveL Offs(pOrigin,258.08,315.04,0.00),v40,z0,tPen\WObj:=wPaper;
    MoveL Offs(pOrigin,256.80,314.68,0.00),v40,z0,tPen\WObj:=wPaper;
    MoveL Offs(pOrigin,254.68,312.77,0.00),v40,z0,tPen\WObj:=wPaper;
    MoveL Offs(pOrigin,253.19,312.27,0.00),v40,z0,tPen\WObj:=wPaper;
    MoveL Offs(pOrigin,252.55,312.49,0.00),v40,z0,tPen\WObj:=wPaper;
    MoveL Offs(pOrigin,251.70,312.42,0.00),v40,z0,tPen\WObj:=wPaper;
    MoveL Offs(pOrigin,250.92,313.12,0.00),v40,z0,tPen\WObj:=wPaper;
    MoveL Offs(pOrigin,251.06,315.46,0.00),v40,fine,tPen\WObj:=wPaper;
    MoveL Offs(pOrigin,251.06,315.46,6.00),v60,z5,tPen\WObj:=wPaper;
    MoveL Offs(pOrigin,252.34,317.16,6.00),vTravel,z5,tPen\WObj:=wPaper;
    MoveL Offs(pOrigin,252.34,317.16,0.00),v60,z0,tPen\WObj:=wPaper;
    MoveL Offs(pOrigin,252.12,319.08,0.00),v40,z0,tPen\WObj:=wPaper;
    MoveL Offs(pOrigin,252.12,319.08,0.00),v40,z0,tPen\WObj:=wPaper;
    MoveL Offs(pOrigin,252.55,319.85,0.00),v40,z0,tPen\WObj:=wPaper;
    MoveL Offs(pOrigin,254.68,321.20,0.00),v40,z0,tPen\WObj:=wPaper;
    MoveL Offs(pOrigin,255.52,322.26,0.00),v40,fine,tPen\WObj:=wPaper;
    MoveL Offs(pOrigin,255.52,322.26,6.00),v60,z5,tPen\WObj:=wPaper;
    MoveL Offs(pOrigin,256.80,322.69,6.00),vTravel,z5,tPen\WObj:=wPaper;
    MoveL Offs(pOrigin,256.80,322.69,0.00),v60,z0,tPen\WObj:=wPaper;
    MoveL Offs(pOrigin,255.60,322.48,0.00),v40,z0,tPen\WObj:=wPaper;
    MoveL Offs(pOrigin,256.16,324.17,0.00),v40,z0,tPen\WObj:=wPaper;
    MoveL Offs(pOrigin,255.95,323.75,0.00),v40,z0,tPen\WObj:=wPaper;
    MoveL Offs(pOrigin,256.16,324.17,0.00),v40,z0,tPen\WObj:=wPaper;
    MoveL Offs(pOrigin,255.95,323.75,0.00),v40,fine,tPen\WObj:=wPaper;
    MoveL Offs(pOrigin,255.95,323.75,6.00),v60,z5,tPen\WObj:=wPaper;
    MoveL Offs(pOrigin,257.23,324.39,6.00),vTravel,z5,tPen\WObj:=wPaper;
    MoveL Offs(pOrigin,257.23,324.39,0.00),v60,z0,tPen\WObj:=wPaper;
    MoveL Offs(pOrigin,257.44,324.81,0.00),v40,z0,tPen\WObj:=wPaper;
    MoveL Offs(pOrigin,257.23,324.39,0.00),v40,fine,tPen\WObj:=wPaper;
    MoveL Offs(pOrigin,257.23,324.39,6.00),v60,z5,tPen\WObj:=wPaper;
    MoveL Offs(pOrigin,254.46,324.60,6.00),vTravel,z5,tPen\WObj:=wPaper;
    MoveL Offs(pOrigin,254.46,324.60,0.00),v60,z0,tPen\WObj:=wPaper;
    MoveL Offs(pOrigin,254.68,325.02,0.00),v40,z0,tPen\WObj:=wPaper;
    MoveL Offs(pOrigin,254.46,324.60,0.00),v40,fine,tPen\WObj:=wPaper;
    MoveL Offs(pOrigin,254.46,324.60,6.00),v60,z5,tPen\WObj:=wPaper;
    MoveL Offs(pOrigin,253.19,324.60,6.00),vTravel,z5,tPen\WObj:=wPaper;
    MoveL Offs(pOrigin,253.19,324.60,0.00),v60,z0,tPen\WObj:=wPaper;
    MoveL Offs(pOrigin,253.40,325.02,0.00),v40,z0,tPen\WObj:=wPaper;
    MoveL Offs(pOrigin,253.19,324.60,0.00),v40,fine,tPen\WObj:=wPaper;
    MoveL Offs(pOrigin,253.19,324.60,6.00),v60,z5,tPen\WObj:=wPaper;
    MoveL Offs(pOrigin,252.55,323.11,6.00),vTravel,z5,tPen\WObj:=wPaper;
    MoveL Offs(pOrigin,252.55,323.11,0.00),v60,z0,tPen\WObj:=wPaper;
    MoveL Offs(pOrigin,253.82,326.73,0.00),v40,z0,tPen\WObj:=wPaper;
    MoveL Offs(pOrigin,253.82,328.64,0.00),v40,z0,tPen\WObj:=wPaper;
    MoveL Offs(pOrigin,253.40,330.34,0.00),v40,z0,tPen\WObj:=wPaper;
    MoveL Offs(pOrigin,252.27,332.67,0.00),v40,z0,tPen\WObj:=wPaper;
    MoveL Offs(pOrigin,250.85,334.09,0.00),v40,z0,tPen\WObj:=wPaper;
    MoveL Offs(pOrigin,249.57,334.59,0.00),v40,z0,tPen\WObj:=wPaper;
    MoveL Offs(pOrigin,249.15,333.95,0.00),v40,z0,tPen\WObj:=wPaper;
    MoveL Offs(pOrigin,249.15,333.95,0.00),v40,z0,tPen\WObj:=wPaper;
    MoveL Offs(pOrigin,248.94,332.89,0.00),v40,z0,tPen\WObj:=wPaper;
    MoveL Offs(pOrigin,250.00,329.70,0.00),v40,z0,tPen\WObj:=wPaper;
    MoveL Offs(pOrigin,249.57,328.85,0.00),v40,z0,tPen\WObj:=wPaper;
    MoveL Offs(pOrigin,249.22,326.30,0.00),v40,z0,tPen\WObj:=wPaper;
    MoveL Offs(pOrigin,248.16,325.02,0.00),v40,z0,tPen\WObj:=wPaper;
    MoveL Offs(pOrigin,248.09,324.17,0.00),v40,z0,tPen\WObj:=wPaper;
    MoveL Offs(pOrigin,248.09,324.17,0.00),v40,z0,tPen\WObj:=wPaper;
    MoveL Offs(pOrigin,248.09,323.75,0.00),v40,z0,tPen\WObj:=wPaper;
    MoveL Offs(pOrigin,248.51,323.54,0.00),v40,z0,tPen\WObj:=wPaper;
    MoveL Offs(pOrigin,248.09,324.17,0.00),v40,z0,tPen\WObj:=wPaper;
    MoveL Offs(pOrigin,246.39,323.75,0.00),v40,z0,tPen\WObj:=wPaper;
    MoveL Offs(pOrigin,246.39,323.96,0.00),v40,z0,tPen\WObj:=wPaper;
    MoveL Offs(pOrigin,246.39,323.96,0.00),v40,z0,tPen\WObj:=wPaper;
    MoveL Offs(pOrigin,245.11,322.55,0.00),v40,z0,tPen\WObj:=wPaper;
    MoveL Offs(pOrigin,243.41,322.12,0.00),v40,z0,tPen\WObj:=wPaper;
    MoveL Offs(pOrigin,243.20,322.48,0.00),v40,z0,tPen\WObj:=wPaper;
    MoveL Offs(pOrigin,243.70,323.96,0.00),v40,z0,tPen\WObj:=wPaper;
    MoveL Offs(pOrigin,244.69,325.24,0.00),v40,z0,tPen\WObj:=wPaper;
    MoveL Offs(pOrigin,244.69,325.24,0.00),v40,z0,tPen\WObj:=wPaper;
    MoveL Offs(pOrigin,245.32,328.00,0.00),v40,z0,tPen\WObj:=wPaper;
    MoveL Offs(pOrigin,245.11,332.89,0.00),v40,z0,tPen\WObj:=wPaper;
    MoveL Offs(pOrigin,245.11,332.89,0.00),v40,z0,tPen\WObj:=wPaper;
    MoveL Offs(pOrigin,246.25,331.83,0.00),v40,z0,tPen\WObj:=wPaper;
    MoveL Offs(pOrigin,246.81,329.91,0.00),v40,z0,tPen\WObj:=wPaper;
    MoveL Offs(pOrigin,246.81,328.64,0.00),v40,z0,tPen\WObj:=wPaper;
    MoveL Offs(pOrigin,246.03,326.51,0.00),v40,z0,tPen\WObj:=wPaper;
    MoveL Offs(pOrigin,245.32,325.52,0.00),v40,z0,tPen\WObj:=wPaper;
    MoveL Offs(pOrigin,244.69,325.24,0.00),v40,fine,tPen\WObj:=wPaper;
    MoveL Offs(pOrigin,244.69,325.24,6.00),v60,z5,tPen\WObj:=wPaper;
    MoveL Offs(pOrigin,244.05,326.94,6.00),vTravel,z5,tPen\WObj:=wPaper;
    MoveL Offs(pOrigin,244.05,326.94,0.00),v60,z0,tPen\WObj:=wPaper;
    MoveL Offs(pOrigin,244.26,328.00,0.00),v40,z0,tPen\WObj:=wPaper;
    MoveL Offs(pOrigin,244.05,328.21,0.00),v40,z0,tPen\WObj:=wPaper;
    MoveL Offs(pOrigin,244.05,328.21,0.00),v40,z0,tPen\WObj:=wPaper;
    MoveL Offs(pOrigin,244.26,331.40,0.00),v40,z0,tPen\WObj:=wPaper;
    MoveL Offs(pOrigin,243.91,332.46,0.00),v40,z0,tPen\WObj:=wPaper;
    MoveL Offs(pOrigin,242.00,334.59,0.00),v40,z0,tPen\WObj:=wPaper;
    MoveL Offs(pOrigin,241.50,335.65,0.00),v40,z0,tPen\WObj:=wPaper;
    MoveL Offs(pOrigin,241.50,335.65,0.00),v40,z0,tPen\WObj:=wPaper;
  ENDPROC

  PROC DrawPart34()
    MoveL Offs(pOrigin,237.25,337.21,0.00),v40,z0,tPen\WObj:=wPaper;
    MoveL Offs(pOrigin,236.40,338.41,0.00),v40,z0,tPen\WObj:=wPaper;
    MoveL Offs(pOrigin,236.40,338.41,0.00),v40,z0,tPen\WObj:=wPaper;
    MoveL Offs(pOrigin,235.12,338.84,0.00),v40,z0,tPen\WObj:=wPaper;
    MoveL Offs(pOrigin,232.15,338.84,0.00),v40,z0,tPen\WObj:=wPaper;
    MoveL Offs(pOrigin,231.30,338.41,0.00),v40,z0,tPen\WObj:=wPaper;
    MoveL Offs(pOrigin,228.32,338.41,0.00),v40,z0,tPen\WObj:=wPaper;
    MoveL Offs(pOrigin,227.48,337.99,0.00),v40,z0,tPen\WObj:=wPaper;
    MoveL Offs(pOrigin,227.19,337.35,0.00),v40,z0,tPen\WObj:=wPaper;
    MoveL Offs(pOrigin,229.39,336.71,0.00),v40,z0,tPen\WObj:=wPaper;
    MoveL Offs(pOrigin,234.06,336.29,0.00),v40,z0,tPen\WObj:=wPaper;
    MoveL Offs(pOrigin,237.04,335.37,0.00),v40,z0,tPen\WObj:=wPaper;
    MoveL Offs(pOrigin,237.96,334.80,0.00),v40,z0,tPen\WObj:=wPaper;
    MoveL Offs(pOrigin,238.31,333.31,0.00),v40,z0,tPen\WObj:=wPaper;
    MoveL Offs(pOrigin,238.31,333.31,0.00),v40,z0,tPen\WObj:=wPaper;
    MoveL Offs(pOrigin,240.58,331.75,0.00),v40,z0,tPen\WObj:=wPaper;
    MoveL Offs(pOrigin,240.65,330.76,0.00),v40,z0,tPen\WObj:=wPaper;
    MoveL Offs(pOrigin,240.65,330.76,0.00),v40,z0,tPen\WObj:=wPaper;
    MoveL Offs(pOrigin,241.50,329.70,0.00),v40,z0,tPen\WObj:=wPaper;
    MoveL Offs(pOrigin,241.50,328.00,0.00),v40,z0,tPen\WObj:=wPaper;
    MoveL Offs(pOrigin,241.22,326.94,0.00),v40,z0,tPen\WObj:=wPaper;
    MoveL Offs(pOrigin,239.59,325.88,0.00),v40,z0,tPen\WObj:=wPaper;
    MoveL Offs(pOrigin,239.59,325.88,0.00),v40,z0,tPen\WObj:=wPaper;
    MoveL Offs(pOrigin,239.66,323.33,0.00),v40,z0,tPen\WObj:=wPaper;
    MoveL Offs(pOrigin,240.01,323.18,0.00),v40,z0,tPen\WObj:=wPaper;
    MoveL Offs(pOrigin,241.93,324.60,0.00),v40,z0,tPen\WObj:=wPaper;
    MoveL Offs(pOrigin,243.41,326.94,0.00),v40,z0,tPen\WObj:=wPaper;
    MoveL Offs(pOrigin,244.05,326.94,0.00),v40,z0,tPen\WObj:=wPaper;
    MoveL Offs(pOrigin,243.41,327.15,0.00),v40,z0,tPen\WObj:=wPaper;
    MoveL Offs(pOrigin,243.41,327.58,0.00),v40,z0,tPen\WObj:=wPaper;
    MoveL Offs(pOrigin,244.05,328.21,0.00),v40,fine,tPen\WObj:=wPaper;
    MoveL Offs(pOrigin,244.05,328.21,6.00),v60,z5,tPen\WObj:=wPaper;
    MoveL Offs(pOrigin,240.23,328.00,6.00),vTravel,z5,tPen\WObj:=wPaper;
    MoveL Offs(pOrigin,240.23,328.00,0.00),v60,z0,tPen\WObj:=wPaper;
    MoveL Offs(pOrigin,240.44,330.12,0.00),v40,z0,tPen\WObj:=wPaper;
    MoveL Offs(pOrigin,240.44,330.12,0.00),v40,z0,tPen\WObj:=wPaper;
    MoveL Offs(pOrigin,239.38,330.12,0.00),v40,z0,tPen\WObj:=wPaper;
    MoveL Offs(pOrigin,239.38,330.12,0.00),v40,z0,tPen\WObj:=wPaper;
    MoveL Offs(pOrigin,239.16,331.40,0.00),v40,z0,tPen\WObj:=wPaper;
    MoveL Offs(pOrigin,239.59,332.04,0.00),v40,fine,tPen\WObj:=wPaper;
    MoveL Offs(pOrigin,239.59,332.04,6.00),v60,z5,tPen\WObj:=wPaper;
    MoveL Offs(pOrigin,238.31,333.31,6.00),vTravel,z5,tPen\WObj:=wPaper;
    MoveL Offs(pOrigin,238.31,333.31,0.00),v60,z0,tPen\WObj:=wPaper;
    MoveL Offs(pOrigin,236.82,333.03,0.00),v40,z0,tPen\WObj:=wPaper;
    MoveL Offs(pOrigin,236.61,332.67,0.00),v40,z0,tPen\WObj:=wPaper;
    MoveL Offs(pOrigin,236.90,331.61,0.00),v40,z0,tPen\WObj:=wPaper;
    MoveL Offs(pOrigin,237.53,330.98,0.00),v40,z0,tPen\WObj:=wPaper;
    MoveL Offs(pOrigin,238.10,328.85,0.00),v40,z0,tPen\WObj:=wPaper;
    MoveL Offs(pOrigin,237.89,326.09,0.00),v40,z0,tPen\WObj:=wPaper;
    MoveL Offs(pOrigin,238.10,325.73,0.00),v40,z0,tPen\WObj:=wPaper;
    MoveL Offs(pOrigin,238.74,325.66,0.00),v40,z0,tPen\WObj:=wPaper;
    MoveL Offs(pOrigin,239.80,326.30,0.00),v40,z0,tPen\WObj:=wPaper;
    MoveL Offs(pOrigin,239.80,326.30,0.00),v40,z0,tPen\WObj:=wPaper;
    MoveL Offs(pOrigin,240.44,328.00,0.00),v40,z0,tPen\WObj:=wPaper;
    MoveL Offs(pOrigin,240.23,328.00,0.00),v40,z0,tPen\WObj:=wPaper;
    MoveL Offs(pOrigin,239.38,328.00,0.00),v40,z0,tPen\WObj:=wPaper;
    MoveL Offs(pOrigin,239.38,330.12,0.00),v40,fine,tPen\WObj:=wPaper;
    MoveL Offs(pOrigin,239.38,330.12,6.00),v60,z5,tPen\WObj:=wPaper;
    MoveL Offs(pOrigin,237.46,330.76,6.00),vTravel,z5,tPen\WObj:=wPaper;
    MoveL Offs(pOrigin,237.46,330.76,0.00),v60,z0,tPen\WObj:=wPaper;
    MoveL Offs(pOrigin,237.25,331.19,0.00),v40,z0,tPen\WObj:=wPaper;
    MoveL Offs(pOrigin,237.46,330.76,0.00),v40,fine,tPen\WObj:=wPaper;
    MoveL Offs(pOrigin,237.46,330.76,6.00),v60,z5,tPen\WObj:=wPaper;
    MoveL Offs(pOrigin,236.40,331.40,6.00),vTravel,z5,tPen\WObj:=wPaper;
    MoveL Offs(pOrigin,236.40,331.40,0.00),v60,z0,tPen\WObj:=wPaper;
    MoveL Offs(pOrigin,235.34,331.68,0.00),v40,z0,tPen\WObj:=wPaper;
    MoveL Offs(pOrigin,234.70,332.89,0.00),v40,z0,tPen\WObj:=wPaper;
    MoveL Offs(pOrigin,231.94,334.38,0.00),v40,z0,tPen\WObj:=wPaper;
    MoveL Offs(pOrigin,229.60,334.80,0.00),v40,z0,tPen\WObj:=wPaper;
    MoveL Offs(pOrigin,226.62,334.80,0.00),v40,z0,tPen\WObj:=wPaper;
    MoveL Offs(pOrigin,225.99,334.38,0.00),v40,z0,tPen\WObj:=wPaper;
    MoveL Offs(pOrigin,225.99,334.38,0.00),v40,z0,tPen\WObj:=wPaper;
    MoveL Offs(pOrigin,226.20,334.02,0.00),v40,z0,tPen\WObj:=wPaper;
    MoveL Offs(pOrigin,230.02,332.75,0.00),v40,z0,tPen\WObj:=wPaper;
    MoveL Offs(pOrigin,230.73,331.40,0.00),v40,z0,tPen\WObj:=wPaper;
    MoveL Offs(pOrigin,231.30,331.19,0.00),v40,z0,tPen\WObj:=wPaper;
    MoveL Offs(pOrigin,231.30,331.19,0.00),v40,z0,tPen\WObj:=wPaper;
    MoveL Offs(pOrigin,231.44,330.34,0.00),v40,z0,tPen\WObj:=wPaper;
    MoveL Offs(pOrigin,232.93,328.42,0.00),v40,z0,tPen\WObj:=wPaper;
    MoveL Offs(pOrigin,233.21,327.15,0.00),v40,z0,tPen\WObj:=wPaper;
    MoveL Offs(pOrigin,232.86,325.45,0.00),v40,z0,tPen\WObj:=wPaper;
    MoveL Offs(pOrigin,231.51,323.47,0.00),v40,z0,tPen\WObj:=wPaper;
    MoveL Offs(pOrigin,231.09,323.75,0.00),v40,z0,tPen\WObj:=wPaper;
    MoveL Offs(pOrigin,231.30,327.15,0.00),v40,z0,tPen\WObj:=wPaper;
    MoveL Offs(pOrigin,230.73,329.06,0.00),v40,z0,tPen\WObj:=wPaper;
    MoveL Offs(pOrigin,229.81,330.55,0.00),v40,z0,tPen\WObj:=wPaper;
    MoveL Offs(pOrigin,230.02,331.12,0.00),v40,z0,tPen\WObj:=wPaper;
    MoveL Offs(pOrigin,230.66,331.19,0.00),v40,z0,tPen\WObj:=wPaper;
    MoveL Offs(pOrigin,231.30,331.19,0.00),v40,z0,tPen\WObj:=wPaper;
    MoveL Offs(pOrigin,232.36,331.05,0.00),v40,z0,tPen\WObj:=wPaper;
    MoveL Offs(pOrigin,233.00,330.55,0.00),v40,z0,tPen\WObj:=wPaper;
    MoveL Offs(pOrigin,234.06,328.21,0.00),v40,z0,tPen\WObj:=wPaper;
    MoveL Offs(pOrigin,234.06,325.66,0.00),v40,z0,tPen\WObj:=wPaper;
    MoveL Offs(pOrigin,233.43,323.75,0.00),v40,z0,tPen\WObj:=wPaper;
    MoveL Offs(pOrigin,233.50,323.33,0.00),v40,z0,tPen\WObj:=wPaper;
    MoveL Offs(pOrigin,233.85,323.25,0.00),v40,z0,tPen\WObj:=wPaper;
    MoveL Offs(pOrigin,235.55,324.81,0.00),v40,z0,tPen\WObj:=wPaper;
    MoveL Offs(pOrigin,236.61,326.73,0.00),v40,z0,tPen\WObj:=wPaper;
    MoveL Offs(pOrigin,237.04,329.06,0.00),v40,z0,tPen\WObj:=wPaper;
    MoveL Offs(pOrigin,236.40,331.40,0.00),v40,fine,tPen\WObj:=wPaper;
    MoveL Offs(pOrigin,236.40,331.40,6.00),v60,z5,tPen\WObj:=wPaper;
    MoveL Offs(pOrigin,236.61,333.10,6.00),vTravel,z5,tPen\WObj:=wPaper;
    MoveL Offs(pOrigin,236.61,333.10,0.00),v60,z0,tPen\WObj:=wPaper;
    MoveL Offs(pOrigin,235.34,334.02,0.00),v40,z0,tPen\WObj:=wPaper;
    MoveL Offs(pOrigin,232.79,335.01,0.00),v40,fine,tPen\WObj:=wPaper;
    MoveL Offs(pOrigin,232.79,335.01,6.00),v60,z5,tPen\WObj:=wPaper;
    MoveL Offs(pOrigin,229.39,335.65,6.00),vTravel,z5,tPen\WObj:=wPaper;
    MoveL Offs(pOrigin,229.39,335.65,0.00),v60,z0,tPen\WObj:=wPaper;
    MoveL Offs(pOrigin,226.84,335.65,0.00),v40,z0,tPen\WObj:=wPaper;
    MoveL Offs(pOrigin,225.99,336.08,0.00),v40,z0,tPen\WObj:=wPaper;
    MoveL Offs(pOrigin,225.99,336.08,0.00),v40,z0,tPen\WObj:=wPaper;
    MoveL Offs(pOrigin,224.93,335.86,0.00),v40,z0,tPen\WObj:=wPaper;
    MoveL Offs(pOrigin,224.50,335.44,0.00),v40,z0,tPen\WObj:=wPaper;
    MoveL Offs(pOrigin,224.50,334.80,0.00),v40,z0,tPen\WObj:=wPaper;
    MoveL Offs(pOrigin,224.50,334.80,0.00),v40,z0,tPen\WObj:=wPaper;
    MoveL Offs(pOrigin,224.71,334.38,0.00),v40,z0,tPen\WObj:=wPaper;
    MoveL Offs(pOrigin,225.99,334.38,0.00),v40,fine,tPen\WObj:=wPaper;
    MoveL Offs(pOrigin,225.99,334.38,6.00),v60,z5,tPen\WObj:=wPaper;
    MoveL Offs(pOrigin,224.50,334.80,6.00),vTravel,z5,tPen\WObj:=wPaper;
    MoveL Offs(pOrigin,224.50,334.80,0.00),v60,z0,tPen\WObj:=wPaper;
  ENDPROC

